LIN {X 0,Y 312.525,Z 361.177,A -85,B 0,C 180,E1 -15697.386,E2 -15697.386} C_VEL
LIN {X 0,Y 312.489,Z 361.185,A -85,B 0,C 180,E1 -15700.71,E2 -15700.71} C_VEL
LIN {X 0,Y 312.451,Z 361.181,A -85,B 0,C 180,E1 -15704.211,E2 -15704.211} C_VEL
LIN {X 0,Y 312.483,Z 361.184,A -85,B 0,C 180,E1 -15707.92,E2 -15707.92} C_VEL
LIN {X 0,Y 312.498,Z 361.177,A -85,B 0,C 180,E1 -15710.972,E2 -15710.972} C_VEL
LIN {X 0,Y 312.533,Z 361.179,A -85,B 0,C 180,E1 -15714.221,E2 -15714.221} C_VEL
LIN {X 0,Y 312.502,Z 361.178,A -85,B 0,C 180,E1 -15717.334,E2 -15717.334} C_VEL
LIN {X 0,Y 312.521,Z 361.179,A -85,B 0,C 180,E1 -15721.288,E2 -15721.288} C_VEL
LIN {X 0,Y 312.554,Z 361.175,A -85,B 0,C 180,E1 -15724.709,E2 -15724.709} C_VEL
LIN {X 0,Y 312.586,Z 361.17,A -85,B 0,C 180,E1 -15727.53,E2 -15727.53} C_VEL
LIN {X 0,Y 312.554,Z 361.175,A -85,B 0,C 180,E1 -15731.652,E2 -15731.652} C_VEL
LIN {X 0,Y 312.654,Z 361.162,A -85,B 0,C 180,E1 -15735.685,E2 -15735.685} C_VEL
LIN {X 0,Y 312.689,Z 361.158,A -85,B 0,C 180,E1 -15739.642,E2 -15739.642} C_VEL
LIN {X 0,Y 312.799,Z 361.146,A -85,B 0,C 180,E1 -15742.253,E2 -15742.253} C_VEL
LIN {X 0,Y 312.692,Z 361.158,A -85,B 0,C 180,E1 -15744.843,E2 -15744.843} C_VEL
LIN {X 0,Y 312.971,Z 361.126,A -85,B 0,C 180,E1 -15748.714,E2 -15748.714} C_VEL
LIN {X 0,Y 312.978,Z 361.123,A -85,B 0,C 180,E1 -15751.287,E2 -15751.287} C_VEL
LIN {X 0,Y 312.666,Z 361.158,A -85,B 0,C 180,E1 -15753.746,E2 -15753.746} C_VEL
LIN {X 0,Y 313.797,Z 364.207,A -85,B 0,C 180,E1 -15753.98,E2 -15753.98} C_VEL
LIN {X 0,Y 315.109,Z 366.459,A -85,B 0,C 180,E1 -15754.197,E2 -15754.197} C_VEL
LIN {X 0,Y 322.201,Z 378.936,A -85,B 0,C 180,E1 -15755.345,E2 -15755.345} C_VEL
LIN {X 0,Y 335.075,Z 404.668,A -85,B 0,C 180,E1 -15757.378,E2 -15757.378} C_VEL
LIN {X 0,Y 330.989,Z 518.086,A -85,B 0,C 180,E1 -15760.012,E2 -15760.012} C_VEL
LIN {X 0,Y 330.01,Z 533.872,A -85,B 0,C 180,E1 -15760.624,E2 -15760.624} C_VEL
LIN {X 0,Y 328.651,Z 549.395,A -85,B 0,C 180,E1 -15761.487,E2 -15761.487} C_VEL
LIN {X 0,Y 326.95,Z 564.144,A -85,B 0,C 180,E1 -15762.571,E2 -15762.571} C_VEL
LIN {X 0,Y 325.282,Z 576.901,A -85,B 0,C 180,E1 -15763.749,E2 -15763.749} C_VEL
LIN {X 0,Y 323.144,Z 590.398,A -85,B 0,C 180,E1 -15765.278,E2 -15765.278} C_VEL
LIN {X 0,Y 321,Z 602.964,A -85,B 0,C 180,E1 -15767.028,E2 -15767.028} C_VEL
LIN {X 0,Y 318.919,Z 614.479,A -85,B 0,C 180,E1 -15768.977,E2 -15768.977} C_VEL
LIN {X 0,Y 317.03,Z 624.528,A -85,B 0,C 180,E1 -15771.026,E2 -15771.026} C_VEL
LIN {X 0,Y 315.313,Z 633.751,A -85,B 0,C 180,E1 -15773.306,E2 -15773.306} C_VEL
LIN {X 0,Y 313.823,Z 641.736,A -85,B 0,C 180,E1 -15775.715,E2 -15775.715} C_VEL
LIN {X 0,Y 312.703,Z 648.292,A -85,B 0,C 180,E1 -15778.163,E2 -15778.163} C_VEL
LIN {X 0,Y 311.992,Z 652.989,A -85,B 0,C 180,E1 -15780.373,E2 -15780.373} C_VEL
LIN {X 0,Y 311.387,Z 657.033,A -85,B 0,C 180,E1 -15782.799,E2 -15782.799} C_VEL
LIN {X 0,Y 310.853,Z 660.262,A -85,B 0,C 180,E1 -15785.519,E2 -15785.519} C_VEL
LIN {X 0,Y 310.67,Z 661.884,A -85,B 0,C 180,E1 -15787.648,E2 -15787.648} C_VEL
LIN {X 0,Y 310.638,Z 662.675,A -85,B 0,C 180,E1 -15789.714,E2 -15789.714} C_VEL
LIN {X 0,Y 310.68,Z 662.765,A -85,B 0,C 180,E1 -15791.711,E2 -15791.711} C_VEL
LIN {X 0,Y 310.986,Z 661.766,A -85,B 0,C 180,E1 -15794.474,E2 -15794.474} C_VEL
LIN {X 0,Y 311.302,Z 660.45,A -85,B 0,C 180,E1 -15796.257,E2 -15796.257} C_VEL
LIN {X 0,Y 312.085,Z 656.982,A -85,B 0,C 180,E1 -15799.226,E2 -15799.226} C_VEL
LIN {X 0,Y 312.245,Z 656.181,A -85,B 0,C 180,E1 -15799.738,E2 -15799.738} C_VEL
LIN {X 0,Y 311.958,Z 654.592,A -85,B 0,C 180,E1 -15800.782,E2 -15800.782} C_VEL
LIN {X 0,Y 309.828,Z 651.885,A -85,B 0,C 180,E1 -15802.5,E2 -15802.5} C_VEL
LIN {X 0,Y 307.865,Z 648.675,A -85,B 0,C 180,E1 -15804.206,E2 -15804.206} C_VEL
LIN {X 0,Y 307.837,Z 646.264,A -85,B 0,C 180,E1 -15805.211,E2 -15805.211} C_VEL
LIN {X 0,Y 309.567,Z 639.569,A -85,B 0,C 180,E1 -15807.567,E2 -15807.567} C_VEL
LIN {X 0,Y 311.823,Z 630.956,A -85,B 0,C 180,E1 -15810.021,E2 -15810.021} C_VEL
LIN {X 0,Y 314.423,Z 621.191,A -85,B 0,C 180,E1 -15812.277,E2 -15812.277} C_VEL
LIN {X 0,Y 317.078,Z 610.167,A -85,B 0,C 180,E1 -15814.379,E2 -15814.379} C_VEL
LIN {X 0,Y 319.674,Z 598.716,A -85,B 0,C 180,E1 -15816.173,E2 -15816.173} C_VEL
LIN {X 0,Y 322.229,Z 586.6,A -85,B 0,C 180,E1 -15817.73,E2 -15817.73} C_VEL
LIN {X 0,Y 324.848,Z 572.636,A -85,B 0,C 180,E1 -15819.188,E2 -15819.188} C_VEL
LIN {X 0,Y 326.941,Z 558.599,A -85,B 0,C 180,E1 -15820.365,E2 -15820.365} C_VEL
LIN {X 0,Y 328.688,Z 544.34,A -85,B 0,C 180,E1 -15821.292,E2 -15821.292} C_VEL
LIN {X 0,Y 330.129,Z 528.83,A -85,B 0,C 180,E1 -15822.04,E2 -15822.04} C_VEL
LIN {X 0,Y 331.077,Z 513.629,A -85,B 0,C 180,E1 -15822.523,E2 -15822.523} C_VEL
LIN {X 0,Y 335.904,Z 411.379,A -85,B 0,C 180,E1 -15824.997,E2 -15824.997} C_VEL
LIN {X 0,Y 329.841,Z 399.642,A -85,B 0,C 180,E1 -15826.309,E2 -15826.309} C_VEL
LIN {X 0,Y 321.07,Z 385.074,A -85,B 0,C 180,E1 -15828.31,E2 -15828.31} C_VEL
LIN {X 0,Y 314.835,Z 375.782,A -85,B 0,C 180,E1 -15829.839,E2 -15829.839} C_VEL
LIN {X 0,Y 311.604,Z 371.252,A -85,B 0,C 180,E1 -15830.682,E2 -15830.682} C_VEL
LIN {X 0,Y 309.38,Z 367.982,A -85,B 0,C 180,E1 -15831.288,E2 -15831.288} C_VEL
LIN {X 0,Y 308.675,Z 366.924,A -85,B 0,C 180,E1 -15831.487,E2 -15831.487} C_VEL
LIN {X 0,Y 306.652,Z 364.665,A -85,B 0,C 180,E1 -15832.04,E2 -15832.04} C_VEL
LIN {X 0,Y 305.758,Z 362.023,A -85,B 0,C 180,E1 -15832.405,E2 -15832.405} C_VEL
LIN {X 0,Y 305.858,Z 362.008,A -85,B 0,C 180,E1 -15837.366,E2 -15837.366} C_VEL
LIN {X 0,Y 306.012,Z 361.989,A -85,B 0,C 180,E1 -15840,E2 -15840} C_VEL
LIN {X 0,Y 305.882,Z 362.006,A -85,B 0,C 180,E1 -15842.633,E2 -15842.633} C_VEL
LIN {X 0,Y 305.79,Z 362.017,A -85,B 0,C 180,E1 -15846.598,E2 -15846.598} C_VEL
LIN {X 0,Y 305.697,Z 362.029,A -85,B 0,C 180,E1 -15849.26,E2 -15849.26} C_VEL
LIN {X 0,Y 305.589,Z 362.038,A -85,B 0,C 180,E1 -15853.296,E2 -15853.296} C_VEL
LIN {X 0,Y 305.554,Z 362.041,A -85,B 0,C 180,E1 -15856.022,E2 -15856.022} C_VEL
LIN {X 0,Y 305.563,Z 362.043,A -85,B 0,C 180,E1 -15859.436,E2 -15859.436} C_VEL
LIN {X 0,Y 305.493,Z 362.058,A -85,B 0,C 180,E1 -15863.041,E2 -15863.041} C_VEL
LIN {X 0,Y 305.55,Z 362.05,A -85,B 0,C 180,E1 -15866.227,E2 -15866.227} C_VEL
LIN {X 0,Y 305.498,Z 362.054,A -85,B 0,C 180,E1 -15869.049,E2 -15869.049} C_VEL
LIN {X 0,Y 305.467,Z 362.063,A -85,B 0,C 180,E1 -15873.516,E2 -15873.516} C_VEL
LIN {X 0,Y 305.497,Z 362.055,A -85,B 0,C 180,E1 -15876.736,E2 -15876.736} C_VEL
LIN {X 0,Y 305.456,Z 362.063,A -85,B 0,C 180,E1 -15880.599,E2 -15880.599} C_VEL
LIN {X 0,Y 305.453,Z 362.134,A -85,B 0,C 180,E1 -15881.768,E2 -15881.768} C_VEL
LIN {X 0,Y 308.493,Z 370.686,A -85,B 0,C 180,E1 -15885.391,E2 -15885.391} C_VEL
LIN {X 0,Y 311.562,Z 380.053,A -85,B 0,C 180,E1 -15888.832,E2 -15888.832} C_VEL
LIN {X 0,Y 314.609,Z 385.314,A -85,B 0,C 180,E1 -15889.657,E2 -15889.657} C_VEL
LIN {X 0,Y 321.104,Z 396.951,A -85,B 0,C 180,E1 -15891.302,E2 -15891.302} C_VEL
LIN {X 0,Y 327.272,Z 409.327,A -85,B 0,C 180,E1 -15892.78,E2 -15892.78} C_VEL
LIN {X 0,Y 331.591,Z 419.42,A -85,B 0,C 180,E1 -15893.794,E2 -15893.794} C_VEL
LIN {X 0,Y 334.763,Z 442.582,A -85,B 0,C 180,E1 -15894.992,E2 -15894.992} C_VEL
LIN {X 0,Y 329.679,Z 550.26,A -85,B 0,C 180,E1 -15897.614,E2 -15897.614} C_VEL
LIN {X 0,Y 328.139,Z 566.262,A -85,B 0,C 180,E1 -15898.214,E2 -15898.214} C_VEL
LIN {X 0,Y 326.128,Z 581.586,A -85,B 0,C 180,E1 -15899.035,E2 -15899.035} C_VEL
LIN {X 0,Y 323.802,Z 595.93,A -85,B 0,C 180,E1 -15900.052,E2 -15900.052} C_VEL
LIN {X 0,Y 321.345,Z 609.142,A -85,B 0,C 180,E1 -15901.239,E2 -15901.239} C_VEL
LIN {X 0,Y 318.545,Z 622.691,A -85,B 0,C 180,E1 -15902.754,E2 -15902.754} C_VEL
LIN {X 0,Y 315.712,Z 635.085,A -85,B 0,C 180,E1 -15904.449,E2 -15904.449} C_VEL
LIN {X 0,Y 312.807,Z 647.316,A -85,B 0,C 180,E1 -15906.496,E2 -15906.496} C_VEL
LIN {X 0,Y 310.294,Z 658.302,A -85,B 0,C 180,E1 -15908.752,E2 -15908.752} C_VEL
LIN {X 0,Y 308.125,Z 667.5,A -85,B 0,C 180,E1 -15911.032,E2 -15911.032} C_VEL
LIN {X 0,Y 306.463,Z 675.179,A -85,B 0,C 180,E1 -15913.341,E2 -15913.341} C_VEL
LIN {X 0,Y 305.112,Z 682.376,A -85,B 0,C 180,E1 -15916.003,E2 -15916.003} C_VEL
LIN {X 0,Y 304.259,Z 688.089,A -85,B 0,C 180,E1 -15918.676,E2 -15918.676} C_VEL
LIN {X 0,Y 303.897,Z 691.49,A -85,B 0,C 180,E1 -15920.683,E2 -15920.683} C_VEL
LIN {X 0,Y 303.719,Z 694.922,A -85,B 0,C 180,E1 -15923.355,E2 -15923.355} C_VEL
LIN {X 0,Y 303.733,Z 697.078,A -85,B 0,C 180,E1 -15926.019,E2 -15926.019} C_VEL
LIN {X 0,Y 303.826,Z 698.028,A -85,B 0,C 180,E1 -15928.674,E2 -15928.674} C_VEL
LIN {X 0,Y 303.935,Z 698.061,A -85,B 0,C 180,E1 -15929.999,E2 -15929.999} C_VEL
LIN {X 0,Y 303.759,Z 697.203,A -85,B 0,C 180,E1 -15932.652,E2 -15932.652} C_VEL
LIN {X 0,Y 303.722,Z 695.129,A -85,B 0,C 180,E1 -15935.31,E2 -15935.31} C_VEL
LIN {X 0,Y 303.803,Z 691.785,A -85,B 0,C 180,E1 -15937.978,E2 -15937.978} C_VEL
LIN {X 0,Y 304.059,Z 687.063,A -85,B 0,C 180,E1 -15940.655,E2 -15940.655} C_VEL
LIN {X 0,Y 304.782,Z 680.879,A -85,B 0,C 180,E1 -15943.331,E2 -15943.331} C_VEL
LIN {X 0,Y 305.951,Z 673.077,A -85,B 0,C 180,E1 -15946,E2 -15946} C_VEL
LIN {X 0,Y 307.348,Z 664.692,A -85,B 0,C 180,E1 -15948.325,E2 -15948.325} C_VEL
LIN {X 0,Y 309.283,Z 654.625,A -85,B 0,C 180,E1 -15950.622,E2 -15950.622} C_VEL
LIN {X 0,Y 311.152,Z 644.275,A -85,B 0,C 180,E1 -15952.58,E2 -15952.58} C_VEL
LIN {X 0,Y 313.211,Z 633.065,A -85,B 0,C 180,E1 -15954.349,E2 -15954.349} C_VEL
LIN {X 0,Y 315.421,Z 620.977,A -85,B 0,C 180,E1 -15955.929,E2 -15955.929} C_VEL
LIN {X 0,Y 317.659,Z 607.911,A -85,B 0,C 180,E1 -15957.327,E2 -15957.327} C_VEL
LIN {X 0,Y 319.827,Z 593.492,A -85,B 0,C 180,E1 -15958.564,E2 -15958.564} C_VEL
LIN {X 0,Y 321.489,Z 580.177,A -85,B 0,C 180,E1 -15959.463,E2 -15959.463} C_VEL
LIN {X 0,Y 323.084,Z 564.612,A -85,B 0,C 180,E1 -15960.245,E2 -15960.245} C_VEL
LIN {X 0,Y 324.137,Z 549.447,A -85,B 0,C 180,E1 -15960.767,E2 -15960.767} C_VEL
LIN {X 0,Y 328.19,Z 442.647,A -85,B 0,C 180,E1 -15963.277,E2 -15963.277} C_VEL
LIN {X 0,Y 324.682,Z 419.062,A -85,B 0,C 180,E1 -15964.279,E2 -15964.279} C_VEL
LIN {X 0,Y 323.2,Z 411.08,A -85,B 0,C 180,E1 -15964.658,E2 -15964.658} C_VEL
LIN {X 0,Y 314.936,Z 392.022,A -85,B 0,C 180,E1 -15966.101,E2 -15966.101} C_VEL
LIN {X 0,Y 311.738,Z 384.895,A -85,B 0,C 180,E1 -15966.705,E2 -15966.705} C_VEL
LIN {X 0,Y 308.469,Z 372.592,A -85,B 0,C 180,E1 -15969.961,E2 -15969.961} C_VEL
LIN {X 0,Y 305.432,Z 362.068,A -85,B 0,C 180,E1 -15972.973,E2 -15972.973} C_VEL
LIN {X 0,Y 305.456,Z 362.057,A -85,B 0,C 180,E1 -15977.413,E2 -15977.413} C_VEL
LIN {X 0,Y 305.472,Z 362.054,A -85,B 0,C 180,E1 -15981.597,E2 -15981.597} C_VEL
LIN {X 0,Y 305.459,Z 362.065,A -85,B 0,C 180,E1 -15984.887,E2 -15984.887} C_VEL
LIN {X 0,Y 305.448,Z 362.061,A -85,B 0,C 180,E1 -15988.355,E2 -15988.355} C_VEL
LIN {X 0,Y 305.517,Z 362.055,A -85,B 0,C 180,E1 -15991.114,E2 -15991.114} C_VEL
LIN {X 0,Y 305.568,Z 362.043,A -85,B 0,C 180,E1 -15994.088,E2 -15994.088} C_VEL
LIN {X 0,Y 305.497,Z 362.053,A -85,B 0,C 180,E1 -15998.403,E2 -15998.403} C_VEL
LIN {X 0,Y 305.586,Z 362.044,A -85,B 0,C 180,E1 -16001.218,E2 -16001.218} C_VEL
LIN {X 0,Y 305.646,Z 362.036,A -85,B 0,C 180,E1 -16005.349,E2 -16005.349} C_VEL
LIN {X 0,Y 305.635,Z 362.025,A -85,B 0,C 180,E1 -16009.4,E2 -16009.4} C_VEL
LIN {X 0,Y 305.805,Z 362.012,A -85,B 0,C 180,E1 -16012.075,E2 -16012.075} C_VEL
LIN {X 0,Y 305.685,Z 362.033,A -85,B 0,C 180,E1 -16014.724,E2 -16014.724} C_VEL
LIN {X 0,Y 305.955,Z 361.991,A -85,B 0,C 180,E1 -16018.684,E2 -16018.684} C_VEL
LIN {X 0,Y 305.955,Z 361.998,A -85,B 0,C 180,E1 -16021.317,E2 -16021.317} C_VEL
LIN {X 0,Y 305.85,Z 362.005,A -85,B 0,C 180,E1 -16026.598,E2 -16026.598} C_VEL
LIN {X 0,Y 305.734,Z 362.024,A -85,B 0,C 180,E1 -16029.26,E2 -16029.26} C_VEL
LIN {X 0,Y 305.587,Z 362.042,A -85,B 0,C 180,E1 -16033.297,E2 -16033.297} C_VEL
LIN {X 0,Y 305.592,Z 362.034,A -85,B 0,C 180,E1 -16036.021,E2 -16036.021} C_VEL
LIN {X 0,Y 305.574,Z 362.043,A -85,B 0,C 180,E1 -16039.445,E2 -16039.445} C_VEL
LIN {X 0,Y 305.484,Z 362.054,A -85,B 0,C 180,E1 -16043.04,E2 -16043.04} C_VEL
LIN {X 0,Y 305.525,Z 362.041,A -85,B 0,C 180,E1 -16046.22,E2 -16046.22} C_VEL
LIN {X 0,Y 305.495,Z 362.056,A -85,B 0,C 180,E1 -16049.051,E2 -16049.051} C_VEL
LIN {X 0,Y 305.464,Z 362.052,A -85,B 0,C 180,E1 -16053.518,E2 -16053.518} C_VEL
LIN {X 0,Y 305.474,Z 362.056,A -85,B 0,C 180,E1 -16056.74,E2 -16056.74} C_VEL
LIN {X 0,Y 305.454,Z 362.062,A -85,B 0,C 180,E1 -16060.601,E2 -16060.601} C_VEL
LIN {X 0,Y 305.425,Z 362.053,A -85,B 0,C 180,E1 -16063.656,E2 -16063.656} C_VEL
LIN {X 0,Y 305.454,Z 362.059,A -85,B 0,C 180,E1 -16067.415,E2 -16067.415} C_VEL
LIN {X 0,Y 305.467,Z 362.05,A -85,B 0,C 180,E1 -16071.597,E2 -16071.597} C_VEL
LIN {X 0,Y 305.463,Z 362.06,A -85,B 0,C 180,E1 -16074.888,E2 -16074.888} C_VEL
LIN {X 0,Y 305.443,Z 362.058,A -85,B 0,C 180,E1 -16078.359,E2 -16078.359} C_VEL
LIN {X 0,Y 305.488,Z 362.056,A -85,B 0,C 180,E1 -16081.111,E2 -16081.111} C_VEL
LIN {X 0,Y 305.506,Z 362.052,A -85,B 0,C 180,E1 -16084.083,E2 -16084.083} C_VEL
LIN {X 0,Y 305.49,Z 362.056,A -85,B 0,C 180,E1 -16088.403,E2 -16088.403} C_VEL
LIN {X 0,Y 305.512,Z 362.052,A -85,B 0,C 180,E1 -16091.213,E2 -16091.213} C_VEL
LIN {X 0,Y 305.582,Z 362.043,A -85,B 0,C 180,E1 -16095.346,E2 -16095.346} C_VEL
LIN {X 0,Y 305.627,Z 362.037,A -85,B 0,C 180,E1 -16099.4,E2 -16099.4} C_VEL
LIN {X 0,Y 305.75,Z 362.023,A -85,B 0,C 180,E1 -16102.073,E2 -16102.073} C_VEL
LIN {X 0,Y 305.662,Z 362.034,A -85,B 0,C 180,E1 -16104.724,E2 -16104.724} C_VEL
LIN {X 0,Y 305.939,Z 362.002,A -85,B 0,C 180,E1 -16108.684,E2 -16108.684} C_VEL
LIN {X 0,Y 305.946,Z 362,A -85,B 0,C 180,E1 -16111.317,E2 -16111.317} C_VEL
LIN {X 0,Y 305.773,Z 362.014,A -85,B 0,C 180,E1 -16112.932,E2 -16112.932} C_VEL
LIN {X 0,Y 306.841,Z 365.057,A -85,B 0,C 180,E1 -16113.18,E2 -16113.18} C_VEL
LIN {X 0,Y 316.889,Z 382.866,A -85,B 0,C 180,E1 -16114.879,E2 -16114.879} C_VEL
LIN {X 0,Y 328.783,Z 406.691,A -85,B 0,C 180,E1 -16116.808,E2 -16116.808} C_VEL
LIN {X 0,Y 324.637,Z 518.559,A -85,B 0,C 180,E1 -16119.463,E2 -16119.463} C_VEL
LIN {X 0,Y 323.669,Z 533.986,A -85,B 0,C 180,E1 -16120.07,E2 -16120.07} C_VEL
LIN {X 0,Y 322.334,Z 549.035,A -85,B 0,C 180,E1 -16120.913,E2 -16120.913} C_VEL
LIN {X 0,Y 320.545,Z 564.038,A -85,B 0,C 180,E1 -16122.023,E2 -16122.023} C_VEL
LIN {X 0,Y 318.572,Z 578.392,A -85,B 0,C 180,E1 -16123.384,E2 -16123.384} C_VEL
LIN {X 0,Y 316.352,Z 591.876,A -85,B 0,C 180,E1 -16124.967,E2 -16124.967} C_VEL
LIN {X 0,Y 314.197,Z 604.035,A -85,B 0,C 180,E1 -16126.716,E2 -16126.716} C_VEL
LIN {X 0,Y 312.407,Z 613.648,A -85,B 0,C 180,E1 -16128.358,E2 -16128.358} C_VEL
LIN {X 0,Y 310.328,Z 624.354,A -85,B 0,C 180,E1 -16130.551,E2 -16130.551} C_VEL
LIN {X 0,Y 308.577,Z 633.32,A -85,B 0,C 180,E1 -16132.78,E2 -16132.78} C_VEL
LIN {X 0,Y 307.109,Z 640.854,A -85,B 0,C 180,E1 -16135.048,E2 -16135.048} C_VEL
LIN {X 0,Y 305.932,Z 647.161,A -85,B 0,C 180,E1 -16137.352,E2 -16137.352} C_VEL
LIN {X 0,Y 305.111,Z 652.347,A -85,B 0,C 180,E1 -16139.685,E2 -16139.685} C_VEL
LIN {X 0,Y 304.484,Z 656.53,A -85,B 0,C 180,E1 -16142.065,E2 -16142.065} C_VEL
LIN {X 0,Y 304.082,Z 658.757,A -85,B 0,C 180,E1 -16143.69,E2 -16143.69} C_VEL
LIN {X 0,Y 303.717,Z 661.043,A -85,B 0,C 180,E1 -16145.913,E2 -16145.913} C_VEL
LIN {X 0,Y 303.558,Z 662.756,A -85,B 0,C 180,E1 -16148.691,E2 -16148.691} C_VEL
LIN {X 0,Y 303.564,Z 663.194,A -85,B 0,C 180,E1 -16150.41,E2 -16150.41} C_VEL
LIN {X 0,Y 303.632,Z 663.156,A -85,B 0,C 180,E1 -16152.209,E2 -16152.209} C_VEL
LIN {X 0,Y 303.848,Z 662.447,A -85,B 0,C 180,E1 -16154.189,E2 -16154.189} C_VEL
LIN {X 0,Y 304.184,Z 661.159,A -85,B 0,C 180,E1 -16156.121,E2 -16156.121} C_VEL
LIN {X 0,Y 304.647,Z 659.329,A -85,B 0,C 180,E1 -16158.008,E2 -16158.008} C_VEL
LIN {X 0,Y 305.5,Z 655.63,A -85,B 0,C 180,E1 -16160.679,E2 -16160.679} C_VEL
LIN {X 0,Y 306.768,Z 650.421,A -85,B 0,C 180,E1 -16163.44,E2 -16163.44} C_VEL
LIN {X 0,Y 307.837,Z 646.264,A -85,B 0,C 180,E1 -16165.211,E2 -16165.211} C_VEL
LIN {X 0,Y 307.873,Z 643.766,A -85,B 0,C 180,E1 -16166.201,E2 -16166.201} C_VEL
LIN {X 0,Y 306.311,Z 639.635,A -85,B 0,C 180,E1 -16167.855,E2 -16167.855} C_VEL
LIN {X 0,Y 304.897,Z 635.081,A -85,B 0,C 180,E1 -16169.489,E2 -16169.489} C_VEL
LIN {X 0,Y 305.162,Z 631.888,A -85,B 0,C 180,E1 -16170.429,E2 -16170.429} C_VEL
LIN {X 0,Y 308.019,Z 621.685,A -85,B 0,C 180,E1 -16172.856,E2 -16172.856} C_VEL
LIN {X 0,Y 310.803,Z 610.698,A -85,B 0,C 180,E1 -16174.989,E2 -16174.989} C_VEL
LIN {X 0,Y 313.499,Z 599.334,A -85,B 0,C 180,E1 -16176.801,E2 -16176.801} C_VEL
LIN {X 0,Y 316.402,Z 586.157,A -85,B 0,C 180,E1 -16178.512,E2 -16178.512} C_VEL
LIN {X 0,Y 319.042,Z 572.446,A -85,B 0,C 180,E1 -16179.951,E2 -16179.951} C_VEL
LIN {X 0,Y 321.141,Z 559.097,A -85,B 0,C 180,E1 -16181.085,E2 -16181.085} C_VEL
LIN {X 0,Y 323.112,Z 543.453,A -85,B 0,C 180,E1 -16182.107,E2 -16182.107} C_VEL
LIN {X 0,Y 324.532,Z 528.086,A -85,B 0,C 180,E1 -16182.837,E2 -16182.837} C_VEL
LIN {X 0,Y 325.566,Z 512.416,A -85,B 0,C 180,E1 -16183.315,E2 -16183.315} C_VEL
LIN {X 0,Y 330.404,Z 413.808,A -85,B 0,C 180,E1 -16185.752,E2 -16185.752} C_VEL
LIN {X 0,Y 324.344,Z 402.299,A -85,B 0,C 180,E1 -16187.121,E2 -16187.121} C_VEL
LIN {X 0,Y 316.457,Z 389.025,A -85,B 0,C 180,E1 -16189.022,E2 -16189.022} C_VEL
LIN {X 0,Y 310.796,Z 380.655,A -85,B 0,C 180,E1 -16190.475,E2 -16190.475} C_VEL
LIN {X 0,Y 308.04,Z 376.701,A -85,B 0,C 180,E1 -16191.222,E2 -16191.222} C_VEL
LIN {X 0,Y 305.121,Z 372.518,A -85,B 0,C 180,E1 -16192.056,E2 -16192.056} C_VEL
LIN {X 0,Y 302.886,Z 369.527,A -85,B 0,C 180,E1 -16192.709,E2 -16192.709} C_VEL
LIN {X 0,Y 302.03,Z 368.043,A -85,B 0,C 180,E1 -16192.983,E2 -16192.983} C_VEL
LIN {X 0,Y 299.775,Z 365.827,A -85,B 0,C 180,E1 -16193.648,E2 -16193.648} C_VEL
LIN {X 0,Y 298.79,Z 363.526,A -85,B 0,C 180,E1 -16194.008,E2 -16194.008} C_VEL
LIN {X 0,Y 298.67,Z 362.908,A -85,B 0,C 180,E1 -16194.091,E2 -16194.091} C_VEL
LIN {X 0,Y 298.916,Z 362.876,A -85,B 0,C 180,E1 -16198.652,E2 -16198.652} C_VEL
LIN {X 0,Y 298.92,Z 362.873,A -85,B 0,C 180,E1 -16201.347,E2 -16201.347} C_VEL
LIN {X 0,Y 298.638,Z 362.908,A -85,B 0,C 180,E1 -16205.401,E2 -16205.401} C_VEL
LIN {X 0,Y 298.71,Z 362.903,A -85,B 0,C 180,E1 -16208.819,E2 -16208.819} C_VEL
LIN {X 0,Y 298.548,Z 362.917,A -85,B 0,C 180,E1 -16213.615,E2 -16213.615} C_VEL
LIN {X 0,Y 298.489,Z 362.923,A -85,B 0,C 180,E1 -16216.412,E2 -16216.412} C_VEL
LIN {X 0,Y 298.501,Z 362.925,A -85,B 0,C 180,E1 -16219.647,E2 -16219.647} C_VEL
LIN {X 0,Y 298.46,Z 362.93,A -85,B 0,C 180,E1 -16223.597,E2 -16223.597} C_VEL
LIN {X 0,Y 298.491,Z 362.926,A -85,B 0,C 180,E1 -16226.574,E2 -16226.574} C_VEL
LIN {X 0,Y 298.423,Z 362.932,A -85,B 0,C 180,E1 -16229.64,E2 -16229.64} C_VEL
LIN {X 0,Y 298.397,Z 362.937,A -85,B 0,C 180,E1 -16232.799,E2 -16232.799} C_VEL
LIN {X 0,Y 298.466,Z 362.931,A -85,B 0,C 180,E1 -16236.812,E2 -16236.812} C_VEL
LIN {X 0,Y 298.421,Z 362.951,A -85,B 0,C 180,E1 -16240.143,E2 -16240.143} C_VEL
LIN {X 0,Y 301.067,Z 370.515,A -85,B 0,C 180,E1 -16243.642,E2 -16243.642} C_VEL
LIN {X 0,Y 303.349,Z 377.253,A -85,B 0,C 180,E1 -16246.385,E2 -16246.385} C_VEL
LIN {X 0,Y 304.157,Z 379.526,A -85,B 0,C 180,E1 -16247.191,E2 -16247.191} C_VEL
LIN {X 0,Y 307.599,Z 385.003,A -85,B 0,C 180,E1 -16248.194,E2 -16248.194} C_VEL
LIN {X 0,Y 312.48,Z 393.558,A -85,B 0,C 180,E1 -16249.551,E2 -16249.551} C_VEL
LIN {X 0,Y 318.528,Z 404.794,A -85,B 0,C 180,E1 -16251.118,E2 -16251.118} C_VEL
LIN {X 0,Y 324.473,Z 417.574,A -85,B 0,C 180,E1 -16252.601,E2 -16252.601} C_VEL
LIN {X 0,Y 326.593,Z 422.93,A -85,B 0,C 180,E1 -16253.125,E2 -16253.125} C_VEL
LIN {X 0,Y 329.297,Z 443.898,A -85,B 0,C 180,E1 -16254.237,E2 -16254.237} C_VEL
LIN {X 0,Y 324.08,Z 549.494,A -85,B 0,C 180,E1 -16256.845,E2 -16256.845} C_VEL
LIN {X 0,Y 322.452,Z 565.528,A -85,B 0,C 180,E1 -16257.447,E2 -16257.447} C_VEL
LIN {X 0,Y 320.468,Z 580.295,A -85,B 0,C 180,E1 -16258.242,E2 -16258.242} C_VEL
LIN {X 0,Y 317.987,Z 594.759,A -85,B 0,C 180,E1 -16259.262,E2 -16259.262} C_VEL
LIN {X 0,Y 315.17,Z 609.522,A -85,B 0,C 180,E1 -16260.621,E2 -16260.621} C_VEL
LIN {X 0,Y 312.243,Z 622.927,A -85,B 0,C 180,E1 -16262.157,E2 -16262.157} C_VEL
LIN {X 0,Y 309.303,Z 635.222,A -85,B 0,C 180,E1 -16263.88,E2 -16263.88} C_VEL
LIN {X 0,Y 306.704,Z 645.623,A -85,B 0,C 180,E1 -16265.64,E2 -16265.64} C_VEL
LIN {X 0,Y 303.904,Z 656.89,A -85,B 0,C 180,E1 -16267.945,E2 -16267.945} C_VEL
LIN {X 0,Y 301.664,Z 666.142,A -85,B 0,C 180,E1 -16270.256,E2 -16270.256} C_VEL
LIN {X 0,Y 299.584,Z 675.002,A -85,B 0,C 180,E1 -16272.947,E2 -16272.947} C_VEL
LIN {X 0,Y 298.158,Z 682.156,A -85,B 0,C 180,E1 -16275.67,E2 -16275.67} C_VEL
LIN {X 0,Y 297.217,Z 687.815,A -85,B 0,C 180,E1 -16278.404,E2 -16278.404} C_VEL
LIN {X 0,Y 296.828,Z 691.17,A -85,B 0,C 180,E1 -16280.459,E2 -16280.459} C_VEL
LIN {X 0,Y 296.635,Z 694.567,A -85,B 0,C 180,E1 -16283.196,E2 -16283.196} C_VEL
LIN {X 0,Y 296.642,Z 696.707,A -85,B 0,C 180,E1 -16285.924,E2 -16285.924} C_VEL
LIN {X 0,Y 296.732,Z 697.623,A -85,B 0,C 180,E1 -16288.642,E2 -16288.642} C_VEL
LIN {X 0,Y 296.846,Z 697.638,A -85,B 0,C 180,E1 -16289.999,E2 -16289.999} C_VEL
LIN {X 0,Y 296.679,Z 696.742,A -85,B 0,C 180,E1 -16292.715,E2 -16292.715} C_VEL
LIN {X 0,Y 296.64,Z 694.627,A -85,B 0,C 180,E1 -16295.437,E2 -16295.437} C_VEL
LIN {X 0,Y 296.746,Z 691.241,A -85,B 0,C 180,E1 -16298.169,E2 -16298.169} C_VEL
LIN {X 0,Y 297.019,Z 686.483,A -85,B 0,C 180,E1 -16300.911,E2 -16300.911} C_VEL
LIN {X 0,Y 297.792,Z 680.25,A -85,B 0,C 180,E1 -16303.65,E2 -16303.65} C_VEL
LIN {X 0,Y 299.046,Z 672.378,A -85,B 0,C 180,E1 -16306.38,E2 -16306.38} C_VEL
LIN {X 0,Y 300.509,Z 663.943,A -85,B 0,C 180,E1 -16308.757,E2 -16308.757} C_VEL
LIN {X 0,Y 302.555,Z 653.798,A -85,B 0,C 180,E1 -16311.102,E2 -16311.102} C_VEL
LIN {X 0,Y 304.503,Z 643.37,A -85,B 0,C 180,E1 -16313.101,E2 -16313.101} C_VEL
LIN {X 0,Y 306.951,Z 630.979,A -85,B 0,C 180,E1 -16315.06,E2 -16315.06} C_VEL
LIN {X 0,Y 309.277,Z 618.549,A -85,B 0,C 180,E1 -16316.666,E2 -16316.666} C_VEL
LIN {X 0,Y 311.59,Z 605.031,A -85,B 0,C 180,E1 -16318.088,E2 -16318.088} C_VEL
LIN {X 0,Y 313.603,Z 591.232,A -85,B 0,C 180,E1 -16319.253,E2 -16319.253} C_VEL
LIN {X 0,Y 315.407,Z 577.052,A -85,B 0,C 180,E1 -16320.181,E2 -16320.181} C_VEL
LIN {X 0,Y 316.923,Z 562.237,A -85,B 0,C 180,E1 -16320.897,E2 -16320.897} C_VEL
LIN {X 0,Y 317.918,Z 547.341,A -85,B 0,C 180,E1 -16321.391,E2 -16321.391} C_VEL
LIN {X 0,Y 321.999,Z 442.984,A -85,B 0,C 180,E1 -16323.887,E2 -16323.887} C_VEL
LIN {X 0,Y 317.554,Z 414.319,A -85,B 0,C 180,E1 -16325.166,E2 -16325.166} C_VEL
LIN {X 0,Y 309.597,Z 395.873,A -85,B 0,C 180,E1 -16326.591,E2 -16326.591} C_VEL
LIN {X 0,Y 304.386,Z 384.503,A -85,B 0,C 180,E1 -16327.572,E2 -16327.572} C_VEL
LIN {X 0,Y 301.233,Z 372.773,A -85,B 0,C 180,E1 -16330.787,E2 -16330.787} C_VEL
LIN {X 0,Y 298.402,Z 362.944,A -85,B 0,C 180,E1 -16333.71,E2 -16333.71} C_VEL
LIN {X 0,Y 298.399,Z 362.941,A -85,B 0,C 180,E1 -16336.921,E2 -16336.921} C_VEL
LIN {X 0,Y 298.4,Z 362.938,A -85,B 0,C 180,E1 -16341.006,E2 -16341.006} C_VEL
LIN {X 0,Y 298.415,Z 362.94,A -85,B 0,C 180,E1 -16343.93,E2 -16343.93} C_VEL
LIN {X 0,Y 298.392,Z 362.94,A -85,B 0,C 180,E1 -16347.983,E2 -16347.983} C_VEL
LIN {X 0,Y 298.46,Z 362.932,A -85,B 0,C 180,E1 -16351.904,E2 -16351.904} C_VEL
LIN {X 0,Y 298.482,Z 362.929,A -85,B 0,C 180,E1 -16354.924,E2 -16354.924} C_VEL
LIN {X 0,Y 298.446,Z 362.936,A -85,B 0,C 180,E1 -16359.315,E2 -16359.315} C_VEL
LIN {X 0,Y 298.534,Z 362.919,A -85,B 0,C 180,E1 -16362.18,E2 -16362.18} C_VEL
LIN {X 0,Y 298.59,Z 362.918,A -85,B 0,C 180,E1 -16364.995,E2 -16364.995} C_VEL
LIN {X 0,Y 298.59,Z 362.9,A -85,B 0,C 180,E1 -16369.147,E2 -16369.147} C_VEL
LIN {X 0,Y 298.751,Z 362.89,A -85,B 0,C 180,E1 -16371.886,E2 -16371.886} C_VEL
LIN {X 0,Y 298.655,Z 362.908,A -85,B 0,C 180,E1 -16374.599,E2 -16374.599} C_VEL
LIN {X 0,Y 298.921,Z 362.866,A -85,B 0,C 180,E1 -16378.653,E2 -16378.653} C_VEL
LIN {X 0,Y 298.921,Z 362.874,A -85,B 0,C 180,E1 -16381.348,E2 -16381.348} C_VEL
LIN {X 0,Y 298.796,Z 362.882,A -85,B 0,C 180,E1 -16386.754,E2 -16386.754} C_VEL
LIN {X 0,Y 298.678,Z 362.901,A -85,B 0,C 180,E1 -16389.481,E2 -16389.481} C_VEL
LIN {X 0,Y 298.55,Z 362.917,A -85,B 0,C 180,E1 -16393.616,E2 -16393.616} C_VEL
LIN {X 0,Y 298.547,Z 362.911,A -85,B 0,C 180,E1 -16396.409,E2 -16396.409} C_VEL
LIN {X 0,Y 298.508,Z 362.923,A -85,B 0,C 180,E1 -16399.655,E2 -16399.655} C_VEL
LIN {X 0,Y 298.427,Z 362.93,A -85,B 0,C 180,E1 -16403.601,E2 -16403.601} C_VEL
LIN {X 0,Y 298.484,Z 362.919,A -85,B 0,C 180,E1 -16406.576,E2 -16406.576} C_VEL
LIN {X 0,Y 298.42,Z 362.935,A -85,B 0,C 180,E1 -16409.642,E2 -16409.642} C_VEL
LIN {X 0,Y 298.394,Z 362.936,A -85,B 0,C 180,E1 -16412.801,E2 -16412.801} C_VEL
LIN {X 0,Y 298.445,Z 362.931,A -85,B 0,C 180,E1 -16416.808,E2 -16416.808} C_VEL
LIN {X 0,Y 298.386,Z 362.938,A -85,B 0,C 180,E1 -16421.088,E2 -16421.088} C_VEL
LIN {X 0,Y 298.398,Z 362.929,A -85,B 0,C 180,E1 -16423.104,E2 -16423.104} C_VEL
LIN {X 0,Y 298.403,Z 362.94,A -85,B 0,C 180,E1 -16426.922,E2 -16426.922} C_VEL
LIN {X 0,Y 298.399,Z 362.931,A -85,B 0,C 180,E1 -16431.008,E2 -16431.008} C_VEL
LIN {X 0,Y 298.419,Z 362.935,A -85,B 0,C 180,E1 -16433.931,E2 -16433.931} C_VEL
LIN {X 0,Y 298.389,Z 362.936,A -85,B 0,C 180,E1 -16437.986,E2 -16437.986} C_VEL
LIN {X 0,Y 298.424,Z 362.936,A -85,B 0,C 180,E1 -16441.901,E2 -16441.901} C_VEL
LIN {X 0,Y 298.451,Z 362.931,A -85,B 0,C 180,E1 -16444.922,E2 -16444.922} C_VEL
LIN {X 0,Y 298.431,Z 362.929,A -85,B 0,C 180,E1 -16449.315,E2 -16449.315} C_VEL
LIN {X 0,Y 298.451,Z 362.935,A -85,B 0,C 180,E1 -16452.175,E2 -16452.175} C_VEL
LIN {X 0,Y 298.513,Z 362.924,A -85,B 0,C 180,E1 -16454.991,E2 -16454.991} C_VEL
LIN {X 0,Y 298.586,Z 362.915,A -85,B 0,C 180,E1 -16459.147,E2 -16459.147} C_VEL
LIN {X 0,Y 298.701,Z 362.9,A -85,B 0,C 180,E1 -16461.885,E2 -16461.885} C_VEL
LIN {X 0,Y 298.632,Z 362.91,A -85,B 0,C 180,E1 -16464.599,E2 -16464.599} C_VEL
LIN {X 0,Y 298.907,Z 362.879,A -85,B 0,C 180,E1 -16468.653,E2 -16468.653} C_VEL
LIN {X 0,Y 298.842,Z 362.882,A -85,B 0,C 180,E1 -16472.106,E2 -16472.106} C_VEL
LIN {X 0,Y 299.808,Z 365.71,A -85,B 0,C 180,E1 -16472.331,E2 -16472.331} C_VEL
LIN {X 0,Y 311.967,Z 387.524,A -85,B 0,C 180,E1 -16474.462,E2 -16474.462} C_VEL
LIN {X 0,Y 322.521,Z 408.759,A -85,B 0,C 180,E1 -16476.22,E2 -16476.22} C_VEL
LIN {X 0,Y 322.522,Z 412.529,A -85,B 0,C 180,E1 -16476.326,E2 -16476.326} C_VEL
LIN {X 0,Y 318.331,Z 518.965,A -85,B 0,C 180,E1 -16478.891,E2 -16478.891} C_VEL
LIN {X 0,Y 317.277,Z 534.7,A -85,B 0,C 180,E1 -16479.523,E2 -16479.523} C_VEL
LIN {X 0,Y 315.965,Z 549.222,A -85,B 0,C 180,E1 -16480.352,E2 -16480.352} C_VEL
LIN {X 0,Y 314.237,Z 563.519,A -85,B 0,C 180,E1 -16481.417,E2 -16481.417} C_VEL
LIN {X 0,Y 312.108,Z 578.478,A -85,B 0,C 180,E1 -16482.848,E2 -16482.848} C_VEL
LIN {X 0,Y 309.809,Z 591.95,A -85,B 0,C 180,E1 -16484.451,E2 -16484.451} C_VEL
LIN {X 0,Y 307.667,Z 603.691,A -85,B 0,C 180,E1 -16486.155,E2 -16486.155} C_VEL
LIN {X 0,Y 305.535,Z 614.764,A -85,B 0,C 180,E1 -16488.092,E2 -16488.092} C_VEL
LIN {X 0,Y 303.38,Z 625.355,A -85,B 0,C 180,E1 -16490.334,E2 -16490.334} C_VEL
LIN {X 0,Y 301.6,Z 634.24,A -85,B 0,C 180,E1 -16492.613,E2 -16492.613} C_VEL
LIN {X 0,Y 300.079,Z 641.713,A -85,B 0,C 180,E1 -16494.934,E2 -16494.934} C_VEL
LIN {X 0,Y 298.834,Z 648.124,A -85,B 0,C 180,E1 -16497.37,E2 -16497.37} C_VEL
LIN {X 0,Y 298.032,Z 653.047,A -85,B 0,C 180,E1 -16499.684,E2 -16499.684} C_VEL
LIN {X 0,Y 297.469,Z 656.567,A -85,B 0,C 180,E1 -16501.729,E2 -16501.729} C_VEL
LIN {X 0,Y 296.812,Z 660.285,A -85,B 0,C 180,E1 -16504.631,E2 -16504.631} C_VEL
LIN {X 0,Y 296.599,Z 661.828,A -85,B 0,C 180,E1 -16506.327,E2 -16506.327} C_VEL
LIN {X 0,Y 296.483,Z 663.089,A -85,B 0,C 180,E1 -16508.532,E2 -16508.532} C_VEL
LIN {X 0,Y 296.492,Z 663.639,A -85,B 0,C 180,E1 -16510.665,E2 -16510.665} C_VEL
LIN {X 0,Y 296.656,Z 663.273,A -85,B 0,C 180,E1 -16513.396,E2 -16513.396} C_VEL
LIN {X 0,Y 296.919,Z 662.403,A -85,B 0,C 180,E1 -16515.243,E2 -16515.243} C_VEL
LIN {X 0,Y 297.324,Z 660.945,A -85,B 0,C 180,E1 -16517.119,E2 -16517.119} C_VEL
LIN {X 0,Y 298.124,Z 657.919,A -85,B 0,C 180,E1 -16519.771,E2 -16519.771} C_VEL
LIN {X 0,Y 299.441,Z 652.694,A -85,B 0,C 180,E1 -16522.94,E2 -16522.94} C_VEL
LIN {X 0,Y 300.938,Z 647.19,A -85,B 0,C 180,E1 -16525.454,E2 -16525.454} C_VEL
LIN {X 0,Y 302.886,Z 640.047,A -85,B 0,C 180,E1 -16528.042,E2 -16528.042} C_VEL
LIN {X 0,Y 305.162,Z 631.888,A -85,B 0,C 180,E1 -16530.429,E2 -16530.429} C_VEL
LIN {X 0,Y 305.486,Z 628.601,A -85,B 0,C 180,E1 -16531.35,E2 -16531.35} C_VEL
LIN {X 0,Y 304.434,Z 623.175,A -85,B 0,C 180,E1 -16532.9,E2 -16532.9} C_VEL
LIN {X 0,Y 303.494,Z 617.362,A -85,B 0,C 180,E1 -16534.399,E2 -16534.399} C_VEL
LIN {X 0,Y 303.971,Z 613.395,A -85,B 0,C 180,E1 -16535.224,E2 -16535.224} C_VEL
LIN {X 0,Y 306.754,Z 602.467,A -85,B 0,C 180,E1 -16537.077,E2 -16537.077} C_VEL
LIN {X 0,Y 309.683,Z 590.08,A -85,B 0,C 180,E1 -16538.801,E2 -16538.801} C_VEL
LIN {X 0,Y 312.455,Z 576.967,A -85,B 0,C 180,E1 -16540.281,E2 -16540.281} C_VEL
LIN {X 0,Y 314.804,Z 563.279,A -85,B 0,C 180,E1 -16541.539,E2 -16541.539} C_VEL
LIN {X 0,Y 316.806,Z 549.389,A -85,B 0,C 180,E1 -16542.538,E2 -16542.538} C_VEL
LIN {X 0,Y 318.453,Z 534.166,A -85,B 0,C 180,E1 -16543.368,E2 -16543.368} C_VEL
LIN {X 0,Y 319.667,Z 518.708,A -85,B 0,C 180,E1 -16543.943,E2 -16543.943} C_VEL
LIN {X 0,Y 325.071,Z 416.497,A -85,B 0,C 180,E1 -16546.517,E2 -16546.517} C_VEL
LIN {X 0,Y 318.729,Z 404.483,A -85,B 0,C 180,E1 -16548.033,E2 -16548.033} C_VEL
LIN {X 0,Y 311.769,Z 392.928,A -85,B 0,C 180,E1 -16549.79,E2 -16549.79} C_VEL
LIN {X 0,Y 304.909,Z 382.593,A -85,B 0,C 180,E1 -16551.674,E2 -16551.674} C_VEL
LIN {X 0,Y 301.497,Z 377.864,A -85,B 0,C 180,E1 -16552.676,E2 -16552.676} C_VEL
LIN {X 0,Y 298.597,Z 373.765,A -85,B 0,C 180,E1 -16553.581,E2 -16553.581} C_VEL
LIN {X 0,Y 296.089,Z 370.631,A -85,B 0,C 180,E1 -16554.381,E2 -16554.381} C_VEL
LIN {X 0,Y 295.441,Z 369.23,A -85,B 0,C 180,E1 -16554.625,E2 -16554.625} C_VEL
LIN {X 0,Y 293.019,Z 367.334,A -85,B 0,C 180,E1 -16555.399,E2 -16555.399} C_VEL
LIN {X 0,Y 291.823,Z 365.144,A -85,B 0,C 180,E1 -16555.856,E2 -16555.856} C_VEL
LIN {X 0,Y 291.533,Z 363.798,A -85,B 0,C 180,E1 -16556.025,E2 -16556.025} C_VEL
LIN {X 0,Y 291.882,Z 363.752,A -85,B 0,C 180,E1 -16558.62,E2 -16558.62} C_VEL
LIN {X 0,Y 291.887,Z 363.748,A -85,B 0,C 180,E1 -16561.379,E2 -16561.379} C_VEL
LIN {X 0,Y 291.607,Z 363.785,A -85,B 0,C 180,E1 -16565.532,E2 -16565.532} C_VEL
LIN {X 0,Y 291.67,Z 363.779,A -85,B 0,C 180,E1 -16568.909,E2 -16568.909} C_VEL
LIN {X 0,Y 291.519,Z 363.791,A -85,B 0,C 180,E1 -16572.531,E2 -16572.531} C_VEL
LIN {X 0,Y 291.509,Z 363.791,A -85,B 0,C 180,E1 -16575.378,E2 -16575.378} C_VEL
LIN {X 0,Y 291.453,Z 363.805,A -85,B 0,C 180,E1 -16579.874,E2 -16579.874} C_VEL
LIN {X 0,Y 291.403,Z 363.805,A -85,B 0,C 180,E1 -16584.205,E2 -16584.205} C_VEL
LIN {X 0,Y 291.425,Z 363.803,A -85,B 0,C 180,E1 -16587.271,E2 -16587.271} C_VEL
LIN {X 0,Y 291.339,Z 363.816,A -85,B 0,C 180,E1 -16590.436,E2 -16590.436} C_VEL
LIN {X 0,Y 291.346,Z 363.822,A -85,B 0,C 180,E1 -16593.698,E2 -16593.698} C_VEL
LIN {X 0,Y 291.395,Z 363.811,A -85,B 0,C 180,E1 -16597.258,E2 -16597.258} C_VEL
LIN {X 0,Y 291.402,Z 363.984,A -85,B 0,C 180,E1 -16598.407,E2 -16598.407} C_VEL
LIN {X 0,Y 294.116,Z 371.443,A -85,B 0,C 180,E1 -16602.204,E2 -16602.204} C_VEL
LIN {X 0,Y 296.684,Z 378.662,A -85,B 0,C 180,E1 -16605.321,E2 -16605.321} C_VEL
LIN {X 0,Y 299.779,Z 383.739,A -85,B 0,C 180,E1 -16606.338,E2 -16606.338} C_VEL
LIN {X 0,Y 304.704,Z 391.674,A -85,B 0,C 180,E1 -16607.833,E2 -16607.833} C_VEL
LIN {X 0,Y 310.094,Z 401.149,A -85,B 0,C 180,E1 -16609.364,E2 -16609.364} C_VEL
LIN {X 0,Y 316.727,Z 414.467,A -85,B 0,C 180,E1 -16611.14,E2 -16611.14} C_VEL
LIN {X 0,Y 321.529,Z 425.732,A -85,B 0,C 180,E1 -16612.39,E2 -16612.39} C_VEL
LIN {X 0,Y 323.956,Z 445.323,A -85,B 0,C 180,E1 -16613.451,E2 -16613.451} C_VEL
LIN {X 0,Y 318.447,Z 549.876,A -85,B 0,C 180,E1 -16616.085,E2 -16616.085} C_VEL
LIN {X 0,Y 316.755,Z 565.621,A -85,B 0,C 180,E1 -16616.691,E2 -16616.691} C_VEL
LIN {X 0,Y 314.499,Z 581.354,A -85,B 0,C 180,E1 -16617.566,E2 -16617.566} C_VEL
LIN {X 0,Y 311.941,Z 595.504,A -85,B 0,C 180,E1 -16618.6,E2 -16618.6} C_VEL
LIN {X 0,Y 309.454,Z 608.158,A -85,B 0,C 180,E1 -16619.781,E2 -16619.781} C_VEL
LIN {X 0,Y 306.281,Z 622.025,A -85,B 0,C 180,E1 -16621.379,E2 -16621.379} C_VEL
LIN {X 0,Y 303.169,Z 634.356,A -85,B 0,C 180,E1 -16623.124,E2 -16623.124} C_VEL
LIN {X 0,Y 300.214,Z 645.705,A -85,B 0,C 180,E1 -16625.078,E2 -16625.078} C_VEL
LIN {X 0,Y 297.215,Z 657.152,A -85,B 0,C 180,E1 -16627.496,E2 -16627.496} C_VEL
LIN {X 0,Y 294.928,Z 666.065,A -85,B 0,C 180,E1 -16629.785,E2 -16629.785} C_VEL
LIN {X 0,Y 292.733,Z 674.823,A -85,B 0,C 180,E1 -16632.536,E2 -16632.536} C_VEL
LIN {X 0,Y 291.196,Z 681.967,A -85,B 0,C 180,E1 -16635.338,E2 -16635.338} C_VEL
LIN {X 0,Y 290.194,Z 687.553,A -85,B 0,C 180,E1 -16638.12,E2 -16638.12} C_VEL
LIN {X 0,Y 289.751,Z 690.862,A -85,B 0,C 180,E1 -16640.224,E2 -16640.224} C_VEL
LIN {X 0,Y 289.552,Z 694.218,A -85,B 0,C 180,E1 -16643.029,E2 -16643.029} C_VEL
LIN {X 0,Y 289.554,Z 696.338,A -85,B 0,C 180,E1 -16645.824,E2 -16645.824} C_VEL
LIN {X 0,Y 289.64,Z 697.218,A -85,B 0,C 180,E1 -16648.609,E2 -16648.609} C_VEL
LIN {X 0,Y 289.757,Z 697.216,A -85,B 0,C 180,E1 -16649.999,E2 -16649.999} C_VEL
LIN {X 0,Y 289.599,Z 696.281,A -85,B 0,C 180,E1 -16652.781,E2 -16652.781} C_VEL
LIN {X 0,Y 289.584,Z 693.978,A -85,B 0,C 180,E1 -16655.712,E2 -16655.712} C_VEL
LIN {X 0,Y 289.671,Z 690.692,A -85,B 0,C 180,E1 -16658.37,E2 -16658.37} C_VEL
LIN {X 0,Y 289.98,Z 685.891,A -85,B 0,C 180,E1 -16661.179,E2 -16661.179} C_VEL
LIN {X 0,Y 290.819,Z 679.609,A -85,B 0,C 180,E1 -16663.984,E2 -16663.984} C_VEL
LIN {X 0,Y 292.144,Z 671.667,A -85,B 0,C 180,E1 -16666.778,E2 -16666.778} C_VEL
LIN {X 0,Y 293.707,Z 663.181,A -85,B 0,C 180,E1 -16669.209,E2 -16669.209} C_VEL
LIN {X 0,Y 295.848,Z 652.946,A -85,B 0,C 180,E1 -16671.604,E2 -16671.604} C_VEL
LIN {X 0,Y 297.896,Z 642.45,A -85,B 0,C 180,E1 -16673.644,E2 -16673.644} C_VEL
LIN {X 0,Y 300.225,Z 631.045,A -85,B 0,C 180,E1 -16675.476,E2 -16675.476} C_VEL
LIN {X 0,Y 302.607,Z 618.691,A -85,B 0,C 180,E1 -16677.115,E2 -16677.115} C_VEL
LIN {X 0,Y 305,Z 605.284,A -85,B 0,C 180,E1 -16678.563,E2 -16678.563} C_VEL
LIN {X 0,Y 307.276,Z 590.187,A -85,B 0,C 180,E1 -16679.864,E2 -16679.864} C_VEL
LIN {X 0,Y 309.216,Z 575.099,A -85,B 0,C 180,E1 -16680.85,E2 -16680.85} C_VEL
LIN {X 0,Y 310.777,Z 559.674,A -85,B 0,C 180,E1 -16681.577,E2 -16681.577} C_VEL
LIN {X 0,Y 311.778,Z 543.415,A -85,B 0,C 180,E1 -16682.082,E2 -16682.082} C_VEL
LIN {X 0,Y 315.76,Z 443.617,A -85,B 0,C 180,E1 -16684.511,E2 -16684.511} C_VEL
LIN {X 0,Y 311.565,Z 416.621,A -85,B 0,C 180,E1 -16685.75,E2 -16685.75} C_VEL
LIN {X 0,Y 302.863,Z 396.546,A -85,B 0,C 180,E1 -16687.366,E2 -16687.366} C_VEL
LIN {X 0,Y 296.969,Z 383.956,A -85,B 0,C 180,E1 -16688.533,E2 -16688.533} C_VEL
LIN {X 0,Y 293.969,Z 372.956,A -85,B 0,C 180,E1 -16691.661,E2 -16691.661} C_VEL
LIN {X 0,Y 291.339,Z 363.817,A -85,B 0,C 180,E1 -16694.451,E2 -16694.451} C_VEL
LIN {X 0,Y 291.323,Z 363.814,A -85,B 0,C 180,E1 -16698.404,E2 -16698.404} C_VEL
LIN {X 0,Y 291.349,Z 363.814,A -85,B 0,C 180,E1 -16701.158,E2 -16701.158} C_VEL
LIN {X 0,Y 291.358,Z 363.82,A -85,B 0,C 180,E1 -16704.626,E2 -16704.626} C_VEL
LIN {X 0,Y 291.368,Z 363.815,A -85,B 0,C 180,E1 -16707.951,E2 -16707.951} C_VEL
LIN {X 0,Y 291.379,Z 363.816,A -85,B 0,C 180,E1 -16711.158,E2 -16711.158} C_VEL
LIN {X 0,Y 291.413,Z 363.806,A -85,B 0,C 180,E1 -16714.272,E2 -16714.272} C_VEL
LIN {X 0,Y 291.378,Z 363.813,A -85,B 0,C 180,E1 -16717.3,E2 -16717.3} C_VEL
LIN {X 0,Y 291.454,Z 363.804,A -85,B 0,C 180,E1 -16720.27,E2 -16720.27} C_VEL
LIN {X 0,Y 291.552,Z 363.794,A -85,B 0,C 180,E1 -16724.624,E2 -16724.624} C_VEL
LIN {X 0,Y 291.533,Z 363.778,A -85,B 0,C 180,E1 -16728.881,E2 -16728.881} C_VEL
LIN {X 0,Y 291.703,Z 363.768,A -85,B 0,C 180,E1 -16731.689,E2 -16731.689} C_VEL
LIN {X 0,Y 291.626,Z 363.783,A -85,B 0,C 180,E1 -16734.469,E2 -16734.469} C_VEL
LIN {X 0,Y 291.887,Z 363.741,A -85,B 0,C 180,E1 -16738.621,E2 -16738.621} C_VEL
LIN {X 0,Y 291.887,Z 363.75,A -85,B 0,C 180,E1 -16741.38,E2 -16741.38} C_VEL
LIN {X 0,Y 291.744,Z 363.758,A -85,B 0,C 180,E1 -16746.918,E2 -16746.918} C_VEL
LIN {X 0,Y 291.627,Z 363.779,A -85,B 0,C 180,E1 -16749.712,E2 -16749.712} C_VEL
LIN {X 0,Y 291.52,Z 363.792,A -85,B 0,C 180,E1 -16753.951,E2 -16753.951} C_VEL
LIN {X 0,Y 291.485,Z 363.79,A -85,B 0,C 180,E1 -16756.819,E2 -16756.819} C_VEL
LIN {X 0,Y 291.449,Z 363.802,A -85,B 0,C 180,E1 -16759.876,E2 -16759.876} C_VEL
LIN {X 0,Y 291.381,Z 363.809,A -85,B 0,C 180,E1 -16764.208,E2 -16764.208} C_VEL
LIN {X 0,Y 291.419,Z 363.803,A -85,B 0,C 180,E1 -16767.272,E2 -16767.272} C_VEL
LIN {X 0,Y 291.336,Z 363.82,A -85,B 0,C 180,E1 -16770.438,E2 -16770.438} C_VEL
LIN {X 0,Y 291.344,Z 363.81,A -85,B 0,C 180,E1 -16773.699,E2 -16773.699} C_VEL
LIN {X 0,Y 291.375,Z 363.812,A -85,B 0,C 180,E1 -16777.255,E2 -16777.255} C_VEL
LIN {X 0,Y 291.332,Z 363.82,A -85,B 0,C 180,E1 -16780.643,E2 -16780.643} C_VEL
LIN {X 0,Y 291.289,Z 363.816,A -85,B 0,C 180,E1 -16784.403,E2 -16784.403} C_VEL
LIN {X 0,Y 291.326,Z 363.823,A -85,B 0,C 180,E1 -16788.405,E2 -16788.405} C_VEL
LIN {X 0,Y 291.348,Z 363.809,A -85,B 0,C 180,E1 -16791.158,E2 -16791.158} C_VEL
LIN {X 0,Y 291.362,Z 363.819,A -85,B 0,C 180,E1 -16794.627,E2 -16794.627} C_VEL
LIN {X 0,Y 291.367,Z 363.81,A -85,B 0,C 180,E1 -16797.951,E2 -16797.951} C_VEL
LIN {X 0,Y 291.353,Z 363.817,A -85,B 0,C 180,E1 -16801.156,E2 -16801.156} C_VEL
LIN {X 0,Y 291.377,Z 363.81,A -85,B 0,C 180,E1 -16804.269,E2 -16804.269} C_VEL
LIN {X 0,Y 291.377,Z 363.813,A -85,B 0,C 180,E1 -16807.3,E2 -16807.3} C_VEL
LIN {X 0,Y 291.408,Z 363.807,A -85,B 0,C 180,E1 -16810.267,E2 -16810.267} C_VEL
LIN {X 0,Y 291.476,Z 363.8,A -85,B 0,C 180,E1 -16814.683,E2 -16814.683} C_VEL
LIN {X 0,Y 291.531,Z 363.795,A -85,B 0,C 180,E1 -16818.881,E2 -16818.881} C_VEL
LIN {X 0,Y 291.655,Z 363.777,A -85,B 0,C 180,E1 -16821.688,E2 -16821.688} C_VEL
LIN {X 0,Y 291.602,Z 363.785,A -85,B 0,C 180,E1 -16824.468,E2 -16824.468} C_VEL
LIN {X 0,Y 291.874,Z 363.755,A -85,B 0,C 180,E1 -16828.621,E2 -16828.621} C_VEL
LIN {X 0,Y 291.857,Z 363.755,A -85,B 0,C 180,E1 -16831.208,E2 -16831.208} C_VEL
LIN {X 0,Y 292.998,Z 366.823,A -85,B 0,C 180,E1 -16831.484,E2 -16831.484} C_VEL
LIN {X 0,Y 298.007,Z 375.866,A -85,B 0,C 180,E1 -16832.425,E2 -16832.425} C_VEL
LIN {X 0,Y 306.708,Z 391.441,A -85,B 0,C 180,E1 -16833.968,E2 -16833.968} C_VEL
LIN {X 0,Y 316.487,Z 411.181,A -85,B 0,C 180,E1 -16835.654,E2 -16835.654} C_VEL
LIN {X 0,Y 311.991,Z 519.612,A -85,B 0,C 180,E1 -16838.315,E2 -16838.315} C_VEL
LIN {X 0,Y 310.931,Z 535.212,A -85,B 0,C 180,E1 -16838.959,E2 -16838.959} C_VEL
LIN {X 0,Y 309.568,Z 549.725,A -85,B 0,C 180,E1 -16839.804,E2 -16839.804} C_VEL
LIN {X 0,Y 307.759,Z 564.137,A -85,B 0,C 180,E1 -16840.899,E2 -16840.899} C_VEL
LIN {X 0,Y 305.679,Z 578.361,A -85,B 0,C 180,E1 -16842.279,E2 -16842.279} C_VEL
LIN {X 0,Y 303.487,Z 590.982,A -85,B 0,C 180,E1 -16843.782,E2 -16843.782} C_VEL
LIN {X 0,Y 301.185,Z 603.245,A -85,B 0,C 180,E1 -16845.566,E2 -16845.566} C_VEL
LIN {X 0,Y 299.072,Z 613.876,A -85,B 0,C 180,E1 -16847.435,E2 -16847.435} C_VEL
LIN {X 0,Y 296.767,Z 624.728,A -85,B 0,C 180,E1 -16849.723,E2 -16849.723} C_VEL
LIN {X 0,Y 294.885,Z 633.675,A -85,B 0,C 180,E1 -16852.024,E2 -16852.024} C_VEL
LIN {X 0,Y 293.287,Z 641.349,A -85,B 0,C 180,E1 -16854.411,E2 -16854.411} C_VEL
LIN {X 0,Y 291.817,Z 648.7,A -85,B 0,C 180,E1 -16857.232,E2 -16857.232} C_VEL
LIN {X 0,Y 290.983,Z 653.584,A -85,B 0,C 180,E1 -16859.599,E2 -16859.599} C_VEL
LIN {X 0,Y 290.272,Z 657.794,A -85,B 0,C 180,E1 -16862.186,E2 -16862.186} C_VEL
LIN {X 0,Y 289.762,Z 660.536,A -85,B 0,C 180,E1 -16864.446,E2 -16864.446} C_VEL
LIN {X 0,Y 289.418,Z 662.907,A -85,B 0,C 180,E1 -16867.379,E2 -16867.379} C_VEL
LIN {X 0,Y 289.375,Z 663.725,A -85,B 0,C 180,E1 -16869.158,E2 -16869.158} C_VEL
LIN {X 0,Y 289.412,Z 664.088,A -85,B 0,C 180,E1 -16871.166,E2 -16871.166} C_VEL
LIN {X 0,Y 289.552,Z 663.786,A -85,B 0,C 180,E1 -16873.267,E2 -16873.267} C_VEL
LIN {X 0,Y 289.866,Z 662.903,A -85,B 0,C 180,E1 -16875.321,E2 -16875.321} C_VEL
LIN {X 0,Y 290.314,Z 661.432,A -85,B 0,C 180,E1 -16877.325,E2 -16877.325} C_VEL
LIN {X 0,Y 290.898,Z 659.351,A -85,B 0,C 180,E1 -16879.283,E2 -16879.283} C_VEL
LIN {X 0,Y 291.873,Z 655.63,A -85,B 0,C 180,E1 -16881.924,E2 -16881.924} C_VEL
LIN {X 0,Y 293.493,Z 649.897,A -85,B 0,C 180,E1 -16884.92,E2 -16884.92} C_VEL
LIN {X 0,Y 295.5,Z 643.128,A -85,B 0,C 180,E1 -16887.647,E2 -16887.647} C_VEL
LIN {X 0,Y 297.528,Z 636.267,A -85,B 0,C 180,E1 -16889.891,E2 -16889.891} C_VEL
LIN {X 0,Y 300.349,Z 626.712,A -85,B 0,C 180,E1 -16892.427,E2 -16892.427} C_VEL
LIN {X 0,Y 303.245,Z 616.31,A -85,B 0,C 180,E1 -16894.672,E2 -16894.672} C_VEL
LIN {X 0,Y 303.971,Z 613.395,A -85,B 0,C 180,E1 -16895.224,E2 -16895.224} C_VEL
LIN {X 0,Y 304.483,Z 609.351,A -85,B 0,C 180,E1 -16896.03,E2 -16896.03} C_VEL
LIN {X 0,Y 303.762,Z 602.797,A -85,B 0,C 180,E1 -16897.428,E2 -16897.428} C_VEL
LIN {X 0,Y 303.078,Z 595.888,A -85,B 0,C 180,E1 -16898.758,E2 -16898.758} C_VEL
LIN {X 0,Y 303.613,Z 591.278,A -85,B 0,C 180,E1 -16899.444,E2 -16899.444} C_VEL
LIN {X 0,Y 306.402,Z 578.676,A -85,B 0,C 180,E1 -16900.913,E2 -16900.913} C_VEL
LIN {X 0,Y 309.007,Z 564.558,A -85,B 0,C 180,E1 -16902.249,E2 -16902.249} C_VEL
LIN {X 0,Y 311.074,Z 551.065,A -85,B 0,C 180,E1 -16903.258,E2 -16903.258} C_VEL
LIN {X 0,Y 312.86,Z 536.03,A -85,B 0,C 180,E1 -16904.11,E2 -16904.11} C_VEL
LIN {X 0,Y 314.138,Z 521.122,A -85,B 0,C 180,E1 -16904.701,E2 -16904.701} C_VEL
LIN {X 0,Y 319.731,Z 419.071,A -85,B 0,C 180,E1 -16907.327,E2 -16907.327} C_VEL
LIN {X 0,Y 313.965,Z 408.252,A -85,B 0,C 180,E1 -16908.776,E2 -16908.776} C_VEL
LIN {X 0,Y 308.105,Z 398.221,A -85,B 0,C 180,E1 -16910.336,E2 -16910.336} C_VEL
LIN {X 0,Y 301.265,Z 387.841,A -85,B 0,C 180,E1 -16912.291,E2 -16912.291} C_VEL
LIN {X 0,Y 298.047,Z 383.254,A -85,B 0,C 180,E1 -16913.282,E2 -16913.282} C_VEL
LIN {X 0,Y 295.256,Z 379.332,A -85,B 0,C 180,E1 -16914.187,E2 -16914.187} C_VEL
LIN {X 0,Y 292.74,Z 375.871,A -85,B 0,C 180,E1 -16915.05,E2 -16915.05} C_VEL
LIN {X 0,Y 289.596,Z 372.421,A -85,B 0,C 180,E1 -16916.136,E2 -16916.136} C_VEL
LIN {X 0,Y 288.24,Z 370.009,A -85,B 0,C 180,E1 -16916.68,E2 -16916.68} C_VEL
LIN {X 0,Y 285.957,Z 367.819,A -85,B 0,C 180,E1 -16917.534,E2 -16917.534} C_VEL
LIN {X 0,Y 284.92,Z 365.478,A -85,B 0,C 180,E1 -16918.012,E2 -16918.012} C_VEL
LIN {X 0,Y 284.786,Z 364.637,A -85,B 0,C 180,E1 -16918.143,E2 -16918.143} C_VEL
LIN {X 0,Y 284.853,Z 364.624,A -85,B 0,C 180,E1 -16921.413,E2 -16921.413} C_VEL
LIN {X 0,Y 284.646,Z 364.647,A -85,B 0,C 180,E1 -16927.091,E2 -16927.091} C_VEL
LIN {X 0,Y 284.517,Z 364.662,A -85,B 0,C 180,E1 -16929.957,E2 -16929.957} C_VEL
LIN {X 0,Y 284.466,Z 364.676,A -85,B 0,C 180,E1 -16934.303,E2 -16934.303} C_VEL
LIN {X 0,Y 284.388,Z 364.677,A -85,B 0,C 180,E1 -16938.739,E2 -16938.739} C_VEL
LIN {X 0,Y 284.369,Z 364.687,A -85,B 0,C 180,E1 -16943.292,E2 -16943.292} C_VEL
LIN {X 0,Y 284.399,Z 364.678,A -85,B 0,C 180,E1 -16947.173,E2 -16947.173} C_VEL
LIN {X 0,Y 284.298,Z 364.699,A -85,B 0,C 180,E1 -16951.274,E2 -16951.274} C_VEL
LIN {X 0,Y 284.363,Z 364.687,A -85,B 0,C 180,E1 -16955.353,E2 -16955.353} C_VEL
LIN {X 0,Y 284.347,Z 364.707,A -85,B 0,C 180,E1 -16956.238,E2 -16956.238} C_VEL
LIN {X 0,Y 286.462,Z 370.555,A -85,B 0,C 180,E1 -16959.633,E2 -16959.633} C_VEL
LIN {X 0,Y 289.021,Z 377.609,A -85,B 0,C 180,E1 -16963.126,E2 -16963.126} C_VEL
LIN {X 0,Y 292.359,Z 382.822,A -85,B 0,C 180,E1 -16964.356,E2 -16964.356} C_VEL
LIN {X 0,Y 293.79,Z 384.988,A -85,B 0,C 180,E1 -16964.859,E2 -16964.859} C_VEL
LIN {X 0,Y 298.195,Z 392.086,A -85,B 0,C 180,E1 -16966.324,E2 -16966.324} C_VEL
LIN {X 0,Y 301.455,Z 397.58,A -85,B 0,C 180,E1 -16967.344,E2 -16967.344} C_VEL
LIN {X 0,Y 306.314,Z 406.338,A -85,B 0,C 180,E1 -16968.785,E2 -16968.785} C_VEL
LIN {X 0,Y 312.424,Z 418.867,A -85,B 0,C 180,E1 -16970.502,E2 -16970.502} C_VEL
LIN {X 0,Y 316.577,Z 428.641,A -85,B 0,C 180,E1 -16971.629,E2 -16971.629} C_VEL
LIN {X 0,Y 318.683,Z 446.856,A -85,B 0,C 180,E1 -16972.641,E2 -16972.641} C_VEL
LIN {X 0,Y 313.05,Z 548.365,A -85,B 0,C 180,E1 -16975.223,E2 -16975.223} C_VEL
LIN {X 0,Y 311.327,Z 564.367,A -85,B 0,C 180,E1 -16975.837,E2 -16975.837} C_VEL
LIN {X 0,Y 308.966,Z 580.223,A -85,B 0,C 180,E1 -16976.717,E2 -16976.717} C_VEL
LIN {X 0,Y 306.339,Z 594.493,A -85,B 0,C 180,E1 -16977.764,E2 -16977.764} C_VEL
LIN {X 0,Y 303.476,Z 608.104,A -85,B 0,C 180,E1 -16979.041,E2 -16979.041} C_VEL
LIN {X 0,Y 300.368,Z 621.197,A -85,B 0,C 180,E1 -16980.57,E2 -16980.57} C_VEL
LIN {X 0,Y 296.857,Z 634.581,A -85,B 0,C 180,E1 -16982.505,E2 -16982.505} C_VEL
LIN {X 0,Y 293.759,Z 645.8,A -85,B 0,C 180,E1 -16984.491,E2 -16984.491} C_VEL
LIN {X 0,Y 290.791,Z 656.621,A -85,B 0,C 180,E1 -16986.836,E2 -16986.836} C_VEL
LIN {X 0,Y 288.229,Z 665.982,A -85,B 0,C 180,E1 -16989.294,E2 -16989.294} C_VEL
LIN {X 0,Y 285.881,Z 674.667,A -85,B 0,C 180,E1 -16992.103,E2 -16992.103} C_VEL
LIN {X 0,Y 284.21,Z 681.946,A -85,B 0,C 180,E1 -16995.068,E2 -16995.068} C_VEL
LIN {X 0,Y 283.187,Z 687.286,A -85,B 0,C 180,E1 -16997.821,E2 -16997.821} C_VEL
LIN {X 0,Y 282.698,Z 690.558,A -85,B 0,C 180,E1 -16999.978,E2 -16999.978} C_VEL
LIN {X 0,Y 282.465,Z 693.871,A -85,B 0,C 180,E1 -17002.853,E2 -17002.853} C_VEL
LIN {X 0,Y 282.472,Z 695.967,A -85,B 0,C 180,E1 -17005.719,E2 -17005.719} C_VEL
LIN {X 0,Y 282.55,Z 696.814,A -85,B 0,C 180,E1 -17008.574,E2 -17008.574} C_VEL
LIN {X 0,Y 282.668,Z 696.79,A -85,B 0,C 180,E1 -17009.999,E2 -17009.999} C_VEL
LIN {X 0,Y 282.522,Z 695.814,A -85,B 0,C 180,E1 -17012.851,E2 -17012.851} C_VEL
LIN {X 0,Y 282.505,Z 693.615,A -85,B 0,C 180,E1 -17015.71,E2 -17015.71} C_VEL
LIN {X 0,Y 282.593,Z 690.13,A -85,B 0,C 180,E1 -17018.581,E2 -17018.581} C_VEL
LIN {X 0,Y 282.947,Z 685.274,A -85,B 0,C 180,E1 -17021.461,E2 -17021.461} C_VEL
LIN {X 0,Y 283.832,Z 678.928,A -85,B 0,C 180,E1 -17024.336,E2 -17024.336} C_VEL
LIN {X 0,Y 285.221,Z 670.909,A -85,B 0,C 180,E1 -17027.198,E2 -17027.198} C_VEL
LIN {X 0,Y 286.917,Z 662.345,A -85,B 0,C 180,E1 -17029.682,E2 -17029.682} C_VEL
LIN {X 0,Y 288.79,Z 653.699,A -85,B 0,C 180,E1 -17031.765,E2 -17031.765} C_VEL
LIN {X 0,Y 290.884,Z 643.287,A -85,B 0,C 180,E1 -17033.871,E2 -17033.871} C_VEL
LIN {X 0,Y 293.2,Z 632.103,A -85,B 0,C 180,E1 -17035.75,E2 -17035.75} C_VEL
LIN {X 0,Y 295.62,Z 620.044,A -85,B 0,C 180,E1 -17037.426,E2 -17037.426} C_VEL
LIN {X 0,Y 298.113,Z 607.031,A -85,B 0,C 180,E1 -17038.899,E2 -17038.899} C_VEL
LIN {X 0,Y 300.37,Z 593.209,A -85,B 0,C 180,E1 -17040.163,E2 -17040.163} C_VEL
LIN {X 0,Y 302.308,Z 579.479,A -85,B 0,C 180,E1 -17041.148,E2 -17041.148} C_VEL
LIN {X 0,Y 303.949,Z 565.013,A -85,B 0,C 180,E1 -17041.932,E2 -17041.932} C_VEL
LIN {X 0,Y 305.171,Z 549.413,A -85,B 0,C 180,E1 -17042.52,E2 -17042.52} C_VEL
LIN {X 0,Y 309.617,Z 445.907,A -85,B 0,C 180,E1 -17045.097,E2 -17045.097} C_VEL
LIN {X 0,Y 306.797,Z 425.633,A -85,B 0,C 180,E1 -17046.016,E2 -17046.016} C_VEL
LIN {X 0,Y 305.603,Z 418.981,A -85,B 0,C 180,E1 -17046.354,E2 -17046.354} C_VEL
LIN {X 0,Y 297.342,Z 399.939,A -85,B 0,C 180,E1 -17047.935,E2 -17047.935} C_VEL
LIN {X 0,Y 289.606,Z 383.479,A -85,B 0,C 180,E1 -17049.515,E2 -17049.515} C_VEL
LIN {X 0,Y 286.647,Z 372.871,A -85,B 0,C 180,E1 -17052.648,E2 -17052.648} C_VEL
LIN {X 0,Y 284.283,Z 364.695,A -85,B 0,C 180,E1 -17055.229,E2 -17055.229} C_VEL
LIN {X 0,Y 284.268,Z 364.692,A -85,B 0,C 180,E1 -17058.124,E2 -17058.124} C_VEL
LIN {X 0,Y 284.319,Z 364.689,A -85,B 0,C 180,E1 -17062.278,E2 -17062.278} C_VEL
LIN {X 0,Y 284.305,Z 364.694,A -85,B 0,C 180,E1 -17065.351,E2 -17065.351} C_VEL
LIN {X 0,Y 284.292,Z 364.698,A -85,B 0,C 180,E1 -17068.726,E2 -17068.726} C_VEL
LIN {X 0,Y 284.394,Z 364.687,A -85,B 0,C 180,E1 -17072.826,E2 -17072.826} C_VEL
LIN {X 0,Y 284.363,Z 364.689,A -85,B 0,C 180,E1 -17076.707,E2 -17076.707} C_VEL
LIN {X 0,Y 284.4,Z 364.682,A -85,B 0,C 180,E1 -17081.262,E2 -17081.262} C_VEL
LIN {X 0,Y 284.489,Z 364.673,A -85,B 0,C 180,E1 -17084.459,E2 -17084.459} C_VEL
LIN {X 0,Y 284.485,Z 364.655,A -85,B 0,C 180,E1 -17088.602,E2 -17088.602} C_VEL
LIN {X 0,Y 284.654,Z 364.647,A -85,B 0,C 180,E1 -17091.481,E2 -17091.481} C_VEL
LIN {X 0,Y 284.596,Z 364.658,A -85,B 0,C 180,E1 -17094.332,E2 -17094.332} C_VEL
LIN {X 0,Y 284.853,Z 364.616,A -85,B 0,C 180,E1 -17098.587,E2 -17098.587} C_VEL
LIN {X 0,Y 284.853,Z 364.626,A -85,B 0,C 180,E1 -17101.414,E2 -17101.414} C_VEL
LIN {X 0,Y 284.696,Z 364.635,A -85,B 0,C 180,E1 -17107.091,E2 -17107.091} C_VEL
LIN {X 0,Y 284.564,Z 364.659,A -85,B 0,C 180,E1 -17109.956,E2 -17109.956} C_VEL
LIN {X 0,Y 284.48,Z 364.67,A -85,B 0,C 180,E1 -17114.303,E2 -17114.303} C_VEL
LIN {X 0,Y 284.424,Z 364.671,A -85,B 0,C 180,E1 -17117.249,E2 -17117.249} C_VEL
LIN {X 0,Y 284.376,Z 364.685,A -85,B 0,C 180,E1 -17120.243,E2 -17120.243} C_VEL
LIN {X 0,Y 284.335,Z 364.679,A -85,B 0,C 180,E1 -17124.848,E2 -17124.848} C_VEL
LIN {X 0,Y 284.329,Z 364.686,A -85,B 0,C 180,E1 -17128.012,E2 -17128.012} C_VEL
LIN {X 0,Y 284.295,Z 364.695,A -85,B 0,C 180,E1 -17131.275,E2 -17131.275} C_VEL
LIN {X 0,Y 284.34,Z 364.68,A -85,B 0,C 180,E1 -17135.349,E2 -17135.349} C_VEL
LIN {X 0,Y 284.311,Z 364.692,A -85,B 0,C 180,E1 -17138.17,E2 -17138.17} C_VEL
LIN {X 0,Y 284.269,Z 364.696,A -85,B 0,C 180,E1 -17142.125,E2 -17142.125} C_VEL
LIN {X 0,Y 284.255,Z 364.699,A -85,B 0,C 180,E1 -17146.19,E2 -17146.19} C_VEL
LIN {X 0,Y 284.307,Z 364.692,A -85,B 0,C 180,E1 -17150.025,E2 -17150.025} C_VEL
LIN {X 0,Y 284.331,Z 364.69,A -85,B 0,C 180,E1 -17153.615,E2 -17153.615} C_VEL
LIN {X 0,Y 284.307,Z 364.689,A -85,B 0,C 180,E1 -17157.191,E2 -17157.191} C_VEL
LIN {X 0,Y 284.342,Z 364.69,A -85,B 0,C 180,E1 -17160.375,E2 -17160.375} C_VEL
LIN {X 0,Y 284.315,Z 364.689,A -85,B 0,C 180,E1 -17163.581,E2 -17163.581} C_VEL
LIN {X 0,Y 284.334,Z 364.693,A -85,B 0,C 180,E1 -17166.705,E2 -17166.705} C_VEL
LIN {X 0,Y 284.379,Z 364.68,A -85,B 0,C 180,E1 -17169.905,E2 -17169.905} C_VEL
LIN {X 0,Y 284.417,Z 364.679,A -85,B 0,C 180,E1 -17174.517,E2 -17174.517} C_VEL
LIN {X 0,Y 284.467,Z 364.673,A -85,B 0,C 180,E1 -17178.601,E2 -17178.601} C_VEL
LIN {X 0,Y 284.612,Z 364.654,A -85,B 0,C 180,E1 -17181.48,E2 -17181.48} C_VEL
LIN {X 0,Y 284.572,Z 364.662,A -85,B 0,C 180,E1 -17184.331,E2 -17184.331} C_VEL
LIN {X 0,Y 284.841,Z 364.631,A -85,B 0,C 180,E1 -17188.587,E2 -17188.587} C_VEL
LIN {X 0,Y 284.826,Z 364.629,A -85,B 0,C 180,E1 -17190.265,E2 -17190.265} C_VEL
LIN {X 0,Y 285.893,Z 367.612,A -85,B 0,C 180,E1 -17190.545,E2 -17190.545} C_VEL
LIN {X 0,Y 287.295,Z 369.722,A -85,B 0,C 180,E1 -17190.809,E2 -17190.809} C_VEL
LIN {X 0,Y 302.001,Z 396.414,A -85,B 0,C 180,E1 -17193.562,E2 -17193.562} C_VEL
LIN {X 0,Y 310.201,Z 413.206,A -85,B 0,C 180,E1 -17195.021,E2 -17195.021} C_VEL
LIN {X 0,Y 305.747,Z 519.724,A -85,B 0,C 180,E1 -17197.699,E2 -17197.699} C_VEL
LIN {X 0,Y 304.63,Z 535.383,A -85,B 0,C 180,E1 -17198.352,E2 -17198.352} C_VEL
LIN {X 0,Y 303.143,Z 550.468,A -85,B 0,C 180,E1 -17199.248,E2 -17199.248} C_VEL
LIN {X 0,Y 301.194,Z 565.409,A -85,B 0,C 180,E1 -17200.419,E2 -17200.419} C_VEL
LIN {X 0,Y 299.271,Z 578.231,A -85,B 0,C 180,E1 -17201.686,E2 -17201.686} C_VEL
LIN {X 0,Y 296.925,Z 591.401,A -85,B 0,C 180,E1 -17203.282,E2 -17203.282} C_VEL
LIN {X 0,Y 294.374,Z 604.406,A -85,B 0,C 180,E1 -17205.226,E2 -17205.226} C_VEL
LIN {X 0,Y 292.214,Z 614.96,A -85,B 0,C 180,E1 -17207.136,E2 -17207.136} C_VEL
LIN {X 0,Y 289.881,Z 625.563,A -85,B 0,C 180,E1 -17209.445,E2 -17209.445} C_VEL
LIN {X 0,Y 287.852,Z 634.828,A -85,B 0,C 180,E1 -17211.907,E2 -17211.907} C_VEL
LIN {X 0,Y 285.999,Z 643.337,A -85,B 0,C 180,E1 -17214.693,E2 -17214.693} C_VEL
LIN {X 0,Y 284.69,Z 649.719,A -85,B 0,C 180,E1 -17217.286,E2 -17217.286} C_VEL
LIN {X 0,Y 283.78,Z 654.822,A -85,B 0,C 180,E1 -17219.91,E2 -17219.91} C_VEL
LIN {X 0,Y 283.106,Z 658.636,A -85,B 0,C 180,E1 -17222.43,E2 -17222.43} C_VEL
LIN {X 0,Y 282.612,Z 661.445,A -85,B 0,C 180,E1 -17224.888,E2 -17224.888} C_VEL
LIN {X 0,Y 282.348,Z 663.191,A -85,B 0,C 180,E1 -17227.2,E2 -17227.2} C_VEL
LIN {X 0,Y 282.298,Z 664.388,A -85,B 0,C 180,E1 -17230.338,E2 -17230.338} C_VEL
LIN {X 0,Y 282.372,Z 664.448,A -85,B 0,C 180,E1 -17232.223,E2 -17232.223} C_VEL
LIN {X 0,Y 282.572,Z 664.012,A -85,B 0,C 180,E1 -17234.14,E2 -17234.14} C_VEL
LIN {X 0,Y 282.924,Z 663.011,A -85,B 0,C 180,E1 -17236.087,E2 -17236.087} C_VEL
LIN {X 0,Y 283.729,Z 660.495,A -85,B 0,C 180,E1 -17239.015,E2 -17239.015} C_VEL
LIN {X 0,Y 284.894,Z 656.391,A -85,B 0,C 180,E1 -17242.131,E2 -17242.131} C_VEL
LIN {X 0,Y 286.473,Z 651.268,A -85,B 0,C 180,E1 -17244.958,E2 -17244.958} C_VEL
LIN {X 0,Y 288.745,Z 643.976,A -85,B 0,C 180,E1 -17248.03,E2 -17248.03} C_VEL
LIN {X 0,Y 291.335,Z 635.548,A -85,B 0,C 180,E1 -17250.806,E2 -17250.806} C_VEL
LIN {X 0,Y 293.897,Z 627.477,A -85,B 0,C 180,E1 -17252.976,E2 -17252.976} C_VEL
LIN {X 0,Y 297.045,Z 616.727,A -85,B 0,C 180,E1 -17255.354,E2 -17255.354} C_VEL
LIN {X 0,Y 300.185,Z 605.051,A -85,B 0,C 180,E1 -17257.457,E2 -17257.457} C_VEL
LIN {X 0,Y 303.068,Z 593.608,A -85,B 0,C 180,E1 -17259.147,E2 -17259.147} C_VEL
LIN {X 0,Y 303.613,Z 591.278,A -85,B 0,C 180,E1 -17259.444,E2 -17259.444} C_VEL
LIN {X 0,Y 304.167,Z 586.577,A -85,B 0,C 180,E1 -17260.109,E2 -17260.109} C_VEL
LIN {X 0,Y 303.573,Z 578.981,A -85,B 0,C 180,E1 -17261.314,E2 -17261.314} C_VEL
LIN {X 0,Y 302.888,Z 571.131,A -85,B 0,C 180,E1 -17262.447,E2 -17262.447} C_VEL
LIN {X 0,Y 303.262,Z 565.985,A -85,B 0,C 180,E1 -17262.987,E2 -17262.987} C_VEL
LIN {X 0,Y 305.527,Z 551.988,A -85,B 0,C 180,E1 -17264.057,E2 -17264.057} C_VEL
LIN {X 0,Y 307.332,Z 537.48,A -85,B 0,C 180,E1 -17264.906,E2 -17264.906} C_VEL
LIN {X 0,Y 308.674,Z 523.242,A -85,B 0,C 180,E1 -17265.495,E2 -17265.495} C_VEL
LIN {X 0,Y 314.635,Z 422.045,A -85,B 0,C 180,E1 -17268.139,E2 -17268.139} C_VEL
LIN {X 0,Y 308.941,Z 411.263,A -85,B 0,C 180,E1 -17269.643,E2 -17269.643} C_VEL
LIN {X 0,Y 302.685,Z 400.688,A -85,B 0,C 180,E1 -17271.407,E2 -17271.407} C_VEL
LIN {X 0,Y 295.27,Z 389.435,A -85,B 0,C 180,E1 -17273.705,E2 -17273.705} C_VEL
LIN {X 0,Y 291.843,Z 384.704,A -85,B 0,C 180,E1 -17274.862,E2 -17274.862} C_VEL
LIN {X 0,Y 289.152,Z 381.103,A -85,B 0,C 180,E1 -17275.818,E2 -17275.818} C_VEL
LIN {X 0,Y 286.602,Z 378.05,A -85,B 0,C 180,E1 -17276.757,E2 -17276.757} C_VEL
LIN {X 0,Y 285.365,Z 376.069,A -85,B 0,C 180,E1 -17277.264,E2 -17277.264} C_VEL
LIN {X 0,Y 282.872,Z 373.155,A -85,B 0,C 180,E1 -17278.264,E2 -17278.264} C_VEL
LIN {X 0,Y 281.814,Z 371.047,A -85,B 0,C 180,E1 -17278.767,E2 -17278.767} C_VEL
LIN {X 0,Y 279.314,Z 369.019,A -85,B 0,C 180,E1 -17279.819,E2 -17279.819} C_VEL
LIN {X 0,Y 278.016,Z 366.51,A -85,B 0,C 180,E1 -17280.497,E2 -17280.497} C_VEL
LIN {X 0,Y 277.826,Z 365.505,A -85,B 0,C 180,E1 -17280.679,E2 -17280.679} C_VEL
LIN {X 0,Y 277.695,Z 365.518,A -85,B 0,C 180,E1 -17282.901,E2 -17282.901} C_VEL
LIN {X 0,Y 277.604,Z 365.524,A -85,B 0,C 180,E1 -17287.272,E2 -17287.272} C_VEL
LIN {X 0,Y 277.46,Z 365.541,A -85,B 0,C 180,E1 -17290.213,E2 -17290.213} C_VEL
LIN {X 0,Y 277.412,Z 365.553,A -85,B 0,C 180,E1 -17294.675,E2 -17294.675} C_VEL
LIN {X 0,Y 277.337,Z 365.557,A -85,B 0,C 180,E1 -17299.234,E2 -17299.234} C_VEL
LIN {X 0,Y 277.322,Z 365.559,A -85,B 0,C 180,E1 -17304.17,E2 -17304.17} C_VEL
LIN {X 0,Y 277.328,Z 365.559,A -85,B 0,C 180,E1 -17307.505,E2 -17307.505} C_VEL
LIN {X 0,Y 277.274,Z 365.568,A -85,B 0,C 180,E1 -17310.481,E2 -17310.481} C_VEL
LIN {X 0,Y 277.257,Z 365.693,A -85,B 0,C 180,E1 -17313.794,E2 -17313.794} C_VEL
LIN {X 0,Y 278.657,Z 369.015,A -85,B 0,C 180,E1 -17316.188,E2 -17316.188} C_VEL
LIN {X 0,Y 280.761,Z 374.865,A -85,B 0,C 180,E1 -17319.665,E2 -17319.665} C_VEL
LIN {X 0,Y 281.521,Z 376.9,A -85,B 0,C 180,E1 -17320.643,E2 -17320.643} C_VEL
LIN {X 0,Y 286.503,Z 384.202,A -85,B 0,C 180,E1 -17322.711,E2 -17322.711} C_VEL
LIN {X 0,Y 290.682,Z 390.702,A -85,B 0,C 180,E1 -17324.277,E2 -17324.277} C_VEL
LIN {X 0,Y 294.824,Z 397.538,A -85,B 0,C 180,E1 -17325.724,E2 -17325.724} C_VEL
LIN {X 0,Y 298.402,Z 403.753,A -85,B 0,C 180,E1 -17326.896,E2 -17326.896} C_VEL
LIN {X 0,Y 303.534,Z 413.5,A -85,B 0,C 180,E1 -17328.481,E2 -17328.481} C_VEL
LIN {X 0,Y 308.52,Z 424.183,A -85,B 0,C 180,E1 -17329.95,E2 -17329.95} C_VEL
LIN {X 0,Y 311.731,Z 431.842,A -85,B 0,C 180,E1 -17330.856,E2 -17330.856} C_VEL
LIN {X 0,Y 313.463,Z 447.583,A -85,B 0,C 180,E1 -17331.756,E2 -17331.756} C_VEL
LIN {X 0,Y 307.655,Z 548.186,A -85,B 0,C 180,E1 -17334.372,E2 -17334.372} C_VEL
LIN {X 0,Y 305.873,Z 564.065,A -85,B 0,C 180,E1 -17334.991,E2 -17334.991} C_VEL
LIN {X 0,Y 303.534,Z 579.326,A -85,B 0,C 180,E1 -17335.841,E2 -17335.841} C_VEL
LIN {X 0,Y 300.816,Z 593.641,A -85,B 0,C 180,E1 -17336.899,E2 -17336.899} C_VEL
LIN {X 0,Y 297.655,Z 607.842,A -85,B 0,C 180,E1 -17338.247,E2 -17338.247} C_VEL
LIN {X 0,Y 294.222,Z 621.561,A -85,B 0,C 180,E1 -17339.892,E2 -17339.892} C_VEL
LIN {X 0,Y 290.881,Z 633.825,A -85,B 0,C 180,E1 -17341.695,E2 -17341.695} C_VEL
LIN {X 0,Y 287.354,Z 645.925,A -85,B 0,C 180,E1 -17343.88,E2 -17343.88} C_VEL
LIN {X 0,Y 284.499,Z 655.835,A -85,B 0,C 180,E1 -17346.065,E2 -17346.065} C_VEL
LIN {X 0,Y 281.56,Z 665.901,A -85,B 0,C 180,E1 -17348.78,E2 -17348.78} C_VEL
LIN {X 0,Y 279.067,Z 674.51,A -85,B 0,C 180,E1 -17351.651,E2 -17351.651} C_VEL
LIN {X 0,Y 277.317,Z 681.468,A -85,B 0,C 180,E1 -17354.553,E2 -17354.553} C_VEL
LIN {X 0,Y 276.194,Z 687.035,A -85,B 0,C 180,E1 -17357.508,E2 -17357.508} C_VEL
LIN {X 0,Y 275.656,Z 690.265,A -85,B 0,C 180,E1 -17359.719,E2 -17359.719} C_VEL
LIN {X 0,Y 275.367,Z 693.526,A -85,B 0,C 180,E1 -17362.668,E2 -17362.668} C_VEL
LIN {X 0,Y 275.372,Z 695.585,A -85,B 0,C 180,E1 -17365.608,E2 -17365.608} C_VEL
LIN {X 0,Y 275.464,Z 696.411,A -85,B 0,C 180,E1 -17368.537,E2 -17368.537} C_VEL
LIN {X 0,Y 275.578,Z 696.365,A -85,B 0,C 180,E1 -17369.999,E2 -17369.999} C_VEL
LIN {X 0,Y 275.446,Z 695.344,A -85,B 0,C 180,E1 -17372.924,E2 -17372.924} C_VEL
LIN {X 0,Y 275.413,Z 693.093,A -85,B 0,C 180,E1 -17375.858,E2 -17375.858} C_VEL
LIN {X 0,Y 275.527,Z 689.556,A -85,B 0,C 180,E1 -17378.803,E2 -17378.803} C_VEL
LIN {X 0,Y 275.926,Z 684.642,A -85,B 0,C 180,E1 -17381.756,E2 -17381.756} C_VEL
LIN {X 0,Y 276.858,Z 678.231,A -85,B 0,C 180,E1 -17384.705,E2 -17384.705} C_VEL
LIN {X 0,Y 278.349,Z 670.143,A -85,B 0,C 180,E1 -17387.636,E2 -17387.636} C_VEL
LIN {X 0,Y 280.172,Z 661.503,A -85,B 0,C 180,E1 -17390.176,E2 -17390.176} C_VEL
LIN {X 0,Y 282.322,Z 651.714,A -85,B 0,C 180,E1 -17392.546,E2 -17392.546} C_VEL
LIN {X 0,Y 284.748,Z 640.373,A -85,B 0,C 180,E1 -17394.808,E2 -17394.808} C_VEL
LIN {X 0,Y 287.044,Z 629.92,A -85,B 0,C 180,E1 -17396.54,E2 -17396.54} C_VEL
LIN {X 0,Y 289.31,Z 618.804,A -85,B 0,C 180,E1 -17398.077,E2 -17398.077} C_VEL
LIN {X 0,Y 291.552,Z 607.189,A -85,B 0,C 180,E1 -17399.415,E2 -17399.415} C_VEL
LIN {X 0,Y 293.888,Z 593.314,A -85,B 0,C 180,E1 -17400.72,E2 -17400.72} C_VEL
LIN {X 0,Y 295.986,Z 578.68,A -85,B 0,C 180,E1 -17401.791,E2 -17401.791} C_VEL
LIN {X 0,Y 297.807,Z 563.199,A -85,B 0,C 180,E1 -17402.621,E2 -17402.621} C_VEL
LIN {X 0,Y 298.993,Z 548.21,A -85,B 0,C 180,E1 -17403.177,E2 -17403.177} C_VEL
LIN {X 0,Y 303.487,Z 445.966,A -85,B 0,C 180,E1 -17405.777,E2 -17405.777} C_VEL
LIN {X 0,Y 299.818,Z 421.697,A -85,B 0,C 180,E1 -17406.952,E2 -17406.952} C_VEL
LIN {X 0,Y 292.045,Z 403.806,A -85,B 0,C 180,E1 -17408.478,E2 -17408.478} C_VEL
LIN {X 0,Y 284.171,Z 387.162,A -85,B 0,C 180,E1 -17410.081,E2 -17410.081} C_VEL
LIN {X 0,Y 282.248,Z 383.056,A -85,B 0,C 180,E1 -17410.532,E2 -17410.532} C_VEL
LIN {X 0,Y 278.955,Z 371.467,A -85,B 0,C 180,E1 -17414.109,E2 -17414.109} C_VEL
LIN {X 0,Y 277.231,Z 365.58,A -85,B 0,C 180,E1 -17416.083,E2 -17416.083} C_VEL
LIN {X 0,Y 277.231,Z 365.576,A -85,B 0,C 180,E1 -17420.672,E2 -17420.672} C_VEL
LIN {X 0,Y 277.281,Z 365.574,A -85,B 0,C 180,E1 -17424.341,E2 -17424.341} C_VEL
LIN {X 0,Y 277.241,Z 365.575,A -85,B 0,C 180,E1 -17427.836,E2 -17427.836} C_VEL
LIN {X 0,Y 277.286,Z 365.571,A -85,B 0,C 180,E1 -17431.213,E2 -17431.213} C_VEL
LIN {X 0,Y 277.31,Z 365.563,A -85,B 0,C 180,E1 -17434.48,E2 -17434.48} C_VEL
LIN {X 0,Y 277.282,Z 365.567,A -85,B 0,C 180,E1 -17437.655,E2 -17437.655} C_VEL
LIN {X 0,Y 277.342,Z 365.565,A -85,B 0,C 180,E1 -17440.766,E2 -17440.766} C_VEL
LIN {X 0,Y 277.432,Z 365.55,A -85,B 0,C 180,E1 -17445.326,E2 -17445.326} C_VEL
LIN {X 0,Y 277.504,Z 365.523,A -85,B 0,C 180,E1 -17449.789,E2 -17449.789} C_VEL
LIN {X 0,Y 277.646,Z 365.521,A -85,B 0,C 180,E1 -17452.729,E2 -17452.729} C_VEL
LIN {X 0,Y 277.819,Z 365.491,A -85,B 0,C 180,E1 -17458.551,E2 -17458.551} C_VEL
LIN {X 0,Y 277.819,Z 365.502,A -85,B 0,C 180,E1 -17461.45,E2 -17461.45} C_VEL
LIN {X 0,Y 277.651,Z 365.511,A -85,B 0,C 180,E1 -17467.272,E2 -17467.272} C_VEL
LIN {X 0,Y 277.505,Z 365.539,A -85,B 0,C 180,E1 -17470.212,E2 -17470.212} C_VEL
LIN {X 0,Y 277.433,Z 365.544,A -85,B 0,C 180,E1 -17474.675,E2 -17474.675} C_VEL
LIN {X 0,Y 277.343,Z 365.561,A -85,B 0,C 180,E1 -17479.235,E2 -17479.235} C_VEL
LIN {X 0,Y 277.29,Z 365.563,A -85,B 0,C 180,E1 -17484.158,E2 -17484.158} C_VEL
LIN {X 0,Y 277.323,Z 365.558,A -85,B 0,C 180,E1 -17487.505,E2 -17487.505} C_VEL
LIN {X 0,Y 277.271,Z 365.573,A -85,B 0,C 180,E1 -17490.482,E2 -17490.482} C_VEL
LIN {X 0,Y 277.246,Z 365.565,A -85,B 0,C 180,E1 -17493.897,E2 -17493.897} C_VEL
LIN {X 0,Y 277.267,Z 365.568,A -85,B 0,C 180,E1 -17497.47,E2 -17497.47} C_VEL
LIN {X 0,Y 277.209,Z 365.574,A -85,B 0,C 180,E1 -17501.237,E2 -17501.237} C_VEL
LIN {X 0,Y 277.2,Z 365.576,A -85,B 0,C 180,E1 -17505.228,E2 -17505.228} C_VEL
LIN {X 0,Y 277.222,Z 365.573,A -85,B 0,C 180,E1 -17509.513,E2 -17509.513} C_VEL
LIN {X 0,Y 277.265,Z 365.566,A -85,B 0,C 180,E1 -17512.531,E2 -17512.531} C_VEL
LIN {X 0,Y 277.247,Z 365.575,A -85,B 0,C 180,E1 -17516.105,E2 -17516.105} C_VEL
LIN {X 0,Y 277.263,Z 365.568,A -85,B 0,C 180,E1 -17519.54,E2 -17519.54} C_VEL
LIN {X 0,Y 277.298,Z 365.564,A -85,B 0,C 180,E1 -17522.858,E2 -17522.858} C_VEL
LIN {X 0,Y 277.289,Z 365.567,A -85,B 0,C 180,E1 -17526.077,E2 -17526.077} C_VEL
LIN {X 0,Y 277.302,Z 365.568,A -85,B 0,C 180,E1 -17530.764,E2 -17530.764} C_VEL
LIN {X 0,Y 277.374,Z 365.557,A -85,B 0,C 180,E1 -17535.323,E2 -17535.323} C_VEL
LIN {X 0,Y 277.458,Z 365.548,A -85,B 0,C 180,E1 -17539.788,E2 -17539.788} C_VEL
LIN {X 0,Y 277.604,Z 365.532,A -85,B 0,C 180,E1 -17542.728,E2 -17542.728} C_VEL
LIN {X 0,Y 277.808,Z 365.506,A -85,B 0,C 180,E1 -17548.551,E2 -17548.551} C_VEL
LIN {X 0,Y 277.816,Z 365.717,A -85,B 0,C 180,E1 -17549.321,E2 -17549.321} C_VEL
LIN {X 0,Y 278.736,Z 368.264,A -85,B 0,C 180,E1 -17549.547,E2 -17549.547} C_VEL
LIN {X 0,Y 280.441,Z 370.97,A -85,B 0,C 180,E1 -17549.888,E2 -17549.888} C_VEL
LIN {X 0,Y 286.266,Z 381.237,A -85,B 0,C 180,E1 -17551.055,E2 -17551.055} C_VEL
LIN {X 0,Y 296.956,Z 400.755,A -85,B 0,C 180,E1 -17553.087,E2 -17553.087} C_VEL
LIN {X 0,Y 304.111,Z 415.471,A -85,B 0,C 180,E1 -17554.392,E2 -17554.392} C_VEL
LIN {X 0,Y 299.539,Z 519.572,A -85,B 0,C 180,E1 -17557.048,E2 -17557.048} C_VEL
LIN {X 0,Y 298.347,Z 535.704,A -85,B 0,C 180,E1 -17557.726,E2 -17557.726} C_VEL
LIN {X 0,Y 296.712,Z 551.463,A -85,B 0,C 180,E1 -17558.685,E2 -17558.685} C_VEL
LIN {X 0,Y 294.918,Z 565.035,A -85,B 0,C 180,E1 -17559.765,E2 -17559.765} C_VEL
LIN {X 0,Y 292.591,Z 579.734,A -85,B 0,C 180,E1 -17561.255,E2 -17561.255} C_VEL
LIN {X 0,Y 290.2,Z 592.714,A -85,B 0,C 180,E1 -17562.885,E2 -17562.885} C_VEL
LIN {X 0,Y 287.815,Z 604.449,A -85,B 0,C 180,E1 -17564.676,E2 -17564.676} C_VEL
LIN {X 0,Y 285.437,Z 615.664,A -85,B 0,C 180,E1 -17566.75,E2 -17566.75} C_VEL
LIN {X 0,Y 283.288,Z 624.988,A -85,B 0,C 180,E1 -17568.816,E2 -17568.816} C_VEL
LIN {X 0,Y 281.193,Z 634.137,A -85,B 0,C 180,E1 -17571.249,E2 -17571.249} C_VEL
LIN {X 0,Y 279.463,Z 641.82,A -85,B 0,C 180,E1 -17573.727,E2 -17573.727} C_VEL
LIN {X 0,Y 278.052,Z 648.267,A -85,B 0,C 180,E1 -17576.253,E2 -17576.253} C_VEL
LIN {X 0,Y 277.017,Z 653.59,A -85,B 0,C 180,E1 -17578.819,E2 -17578.819} C_VEL
LIN {X 0,Y 276.28,Z 657.833,A -85,B 0,C 180,E1 -17581.432,E2 -17581.432} C_VEL
LIN {X 0,Y 275.664,Z 661.094,A -85,B 0,C 180,E1 -17584.118,E2 -17584.118} C_VEL
LIN {X 0,Y 275.372,Z 662.74,A -85,B 0,C 180,E1 -17585.945,E2 -17585.945} C_VEL
LIN {X 0,Y 275.223,Z 663.941,A -85,B 0,C 180,E1 -17587.797,E2 -17587.797} C_VEL
LIN {X 0,Y 275.203,Z 664.737,A -85,B 0,C 180,E1 -17589.992,E2 -17589.992} C_VEL
LIN {X 0,Y 275.298,Z 664.878,A -85,B 0,C 180,E1 -17592.239,E2 -17592.239} C_VEL
LIN {X 0,Y 275.522,Z 664.42,A -85,B 0,C 180,E1 -17594.419,E2 -17594.419} C_VEL
LIN {X 0,Y 276.206,Z 662.583,A -85,B 0,C 180,E1 -17597.554,E2 -17597.554} C_VEL
LIN {X 0,Y 277.24,Z 659.403,A -85,B 0,C 180,E1 -17600.672,E2 -17600.672} C_VEL
LIN {X 0,Y 278.691,Z 654.769,A -85,B 0,C 180,E1 -17603.802,E2 -17603.802} C_VEL
LIN {X 0,Y 280.481,Z 649.337,A -85,B 0,C 180,E1 -17606.546,E2 -17606.546} C_VEL
LIN {X 0,Y 282.797,Z 642.276,A -85,B 0,C 180,E1 -17609.372,E2 -17609.372} C_VEL
LIN {X 0,Y 285.667,Z 633.596,A -85,B 0,C 180,E1 -17612.131,E2 -17612.131} C_VEL
LIN {X 0,Y 288.49,Z 625.005,A -85,B 0,C 180,E1 -17614.34,E2 -17614.34} C_VEL
LIN {X 0,Y 291.621,Z 614.516,A -85,B 0,C 180,E1 -17616.583,E2 -17616.583} C_VEL
LIN {X 0,Y 294.929,Z 602.707,A -85,B 0,C 180,E1 -17618.643,E2 -17618.643} C_VEL
LIN {X 0,Y 297.893,Z 591.317,A -85,B 0,C 180,E1 -17620.273,E2 -17620.273} C_VEL
LIN {X 0,Y 300.886,Z 578.342,A -85,B 0,C 180,E1 -17621.795,E2 -17621.795} C_VEL
LIN {X 0,Y 303.262,Z 565.985,A -85,B 0,C 180,E1 -17622.987,E2 -17622.987} C_VEL
LIN {X 0,Y 303.628,Z 560.735,A -85,B 0,C 180,E1 -17623.512,E2 -17623.512} C_VEL
LIN {X 0,Y 301.821,Z 545.526,A -85,B 0,C 180,E1 -17625.259,E2 -17625.259} C_VEL
LIN {X 0,Y 301.798,Z 540.077,A -85,B 0,C 180,E1 -17625.677,E2 -17625.677} C_VEL
LIN {X 0,Y 301.992,Z 538.193,A -85,B 0,C 180,E1 -17625.772,E2 -17625.772} C_VEL
LIN {X 0,Y 303.469,Z 523.002,A -85,B 0,C 180,E1 -17626.408,E2 -17626.408} C_VEL
LIN {X 0,Y 309.454,Z 424.631,A -85,B 0,C 180,E1 -17629.021,E2 -17629.021} C_VEL
LIN {X 0,Y 302.969,Z 412.408,A -85,B 0,C 180,E1 -17630.856,E2 -17630.856} C_VEL
LIN {X 0,Y 296.932,Z 402.514,A -85,B 0,C 180,E1 -17632.686,E2 -17632.686} C_VEL
LIN {X 0,Y 291.425,Z 394.182,A -85,B 0,C 180,E1 -17634.507,E2 -17634.507} C_VEL
LIN {X 0,Y 288.774,Z 390.419,A -85,B 0,C 180,E1 -17635.45,E2 -17635.45} C_VEL
LIN {X 0,Y 286.338,Z 387.14,A -85,B 0,C 180,E1 -17636.343,E2 -17636.343} C_VEL
LIN {X 0,Y 283.531,Z 383.482,A -85,B 0,C 180,E1 -17637.447,E2 -17637.447} C_VEL
LIN {X 0,Y 282.488,Z 381.975,A -85,B 0,C 180,E1 -17637.883,E2 -17637.883} C_VEL
LIN {X 0,Y 279.975,Z 378.606,A -85,B 0,C 180,E1 -17638.971,E2 -17638.971} C_VEL
LIN {X 0,Y 279.12,Z 377.303,A -85,B 0,C 180,E1 -17639.368,E2 -17639.368} C_VEL
LIN {X 0,Y 276.729,Z 374.899,A -85,B 0,C 180,E1 -17640.454,E2 -17640.454} C_VEL
LIN {X 0,Y 275.216,Z 372.083,A -85,B 0,C 180,E1 -17641.28,E2 -17641.28} C_VEL
LIN {X 0,Y 272.555,Z 370.4,A -85,B 0,C 180,E1 -17642.6,E2 -17642.6} C_VEL
LIN {X 0,Y 270.895,Z 367.963,A -85,B 0,C 180,E1 -17643.625,E2 -17643.625} C_VEL
LIN {X 0,Y 270.449,Z 366.417,A -85,B 0,C 180,E1 -17644.004,E2 -17644.004} C_VEL
LIN {X 0,Y 270.566,Z 366.401,A -85,B 0,C 180,E1 -17647.462,E2 -17647.462} C_VEL
LIN {X 0,Y 270.413,Z 366.42,A -85,B 0,C 180,E1 -17650.482,E2 -17650.482} C_VEL
LIN {X 0,Y 270.38,Z 366.424,A -85,B 0,C 180,E1 -17655.065,E2 -17655.065} C_VEL
LIN {X 0,Y 270.299,Z 366.437,A -85,B 0,C 180,E1 -17659.755,E2 -17659.755} C_VEL
LIN {X 0,Y 270.277,Z 366.436,A -85,B 0,C 180,E1 -17664.585,E2 -17664.585} C_VEL
LIN {X 0,Y 270.274,Z 366.44,A -85,B 0,C 180,E1 -17667.908,E2 -17667.908} C_VEL
LIN {X 0,Y 270.237,Z 366.588,A -85,B 0,C 180,E1 -17670.731,E2 -17670.731} C_VEL
LIN {X 0,Y 272.505,Z 372.441,A -85,B 0,C 180,E1 -17675.47,E2 -17675.47} C_VEL
LIN {X 0,Y 273.805,Z 375.696,A -85,B 0,C 180,E1 -17677.524,E2 -17677.524} C_VEL
LIN {X 0,Y 279.245,Z 383.435,A -85,B 0,C 180,E1 -17680.219,E2 -17680.219} C_VEL
LIN {X 0,Y 283.754,Z 390.247,A -85,B 0,C 180,E1 -17682.167,E2 -17682.167} C_VEL
LIN {X 0,Y 287.564,Z 396.298,A -85,B 0,C 180,E1 -17683.663,E2 -17683.663} C_VEL
LIN {X 0,Y 291.875,Z 403.626,A -85,B 0,C 180,E1 -17685.242,E2 -17685.242} C_VEL
LIN {X 0,Y 296.603,Z 412.143,A -85,B 0,C 180,E1 -17686.834,E2 -17686.834} C_VEL
LIN {X 0,Y 302.421,Z 424.146,A -85,B 0,C 180,E1 -17688.678,E2 -17688.678} C_VEL
LIN {X 0,Y 306.892,Z 434.922,A -85,B 0,C 180,E1 -17690.043,E2 -17690.043} C_VEL
LIN {X 0,Y 308.389,Z 448.745,A -85,B 0,C 180,E1 -17690.86,E2 -17690.86} C_VEL
LIN {X 0,Y 302.331,Z 548.14,A -85,B 0,C 180,E1 -17693.49,E2 -17693.49} C_VEL
LIN {X 0,Y 300.494,Z 563.783,A -85,B 0,C 180,E1 -17694.114,E2 -17694.114} C_VEL
LIN {X 0,Y 297.947,Z 579.531,A -85,B 0,C 180,E1 -17695.006,E2 -17695.006} C_VEL
LIN {X 0,Y 295.322,Z 592.831,A -85,B 0,C 180,E1 -17695.996,E2 -17695.996} C_VEL
LIN {X 0,Y 292.188,Z 606.575,A -85,B 0,C 180,E1 -17697.304,E2 -17697.304} C_VEL
LIN {X 0,Y 288.793,Z 619.656,A -85,B 0,C 180,E1 -17698.859,E2 -17698.859} C_VEL
LIN {X 0,Y 285.237,Z 632.092,A -85,B 0,C 180,E1 -17700.678,E2 -17700.678} C_VEL
LIN {X 0,Y 281.5,Z 644.391,A -85,B 0,C 180,E1 -17702.894,E2 -17702.894} C_VEL
LIN {X 0,Y 278.388,Z 654.456,A -85,B 0,C 180,E1 -17705.116,E2 -17705.116} C_VEL
LIN {X 0,Y 275.633,Z 663.437,A -85,B 0,C 180,E1 -17707.513,E2 -17707.513} C_VEL
LIN {X 0,Y 273.145,Z 671.381,A -85,B 0,C 180,E1 -17710.066,E2 -17710.066} C_VEL
LIN {X 0,Y 271.251,Z 678.026,A -85,B 0,C 180,E1 -17712.664,E2 -17712.664} C_VEL
LIN {X 0,Y 269.711,Z 684.201,A -85,B 0,C 180,E1 -17715.667,E2 -17715.667} C_VEL
LIN {X 0,Y 268.736,Z 689.019,A -85,B 0,C 180,E1 -17718.688,E2 -17718.688} C_VEL
LIN {X 0,Y 268.395,Z 691.74,A -85,B 0,C 180,E1 -17720.96,E2 -17720.96} C_VEL
LIN {X 0,Y 268.29,Z 694.348,A -85,B 0,C 180,E1 -17723.985,E2 -17723.985} C_VEL
LIN {X 0,Y 268.353,Z 695.764,A -85,B 0,C 180,E1 -17726.997,E2 -17726.997} C_VEL
LIN {X 0,Y 268.489,Z 695.94,A -85,B 0,C 180,E1 -17729.999,E2 -17729.999} C_VEL
LIN {X 0,Y 268.372,Z 694.874,A -85,B 0,C 180,E1 -17733.002,E2 -17733.002} C_VEL
LIN {X 0,Y 268.333,Z 692.573,A -85,B 0,C 180,E1 -17736.013,E2 -17736.013} C_VEL
LIN {X 0,Y 268.441,Z 688.981,A -85,B 0,C 180,E1 -17739.037,E2 -17739.037} C_VEL
LIN {X 0,Y 268.922,Z 684.011,A -85,B 0,C 180,E1 -17742.067,E2 -17742.067} C_VEL
LIN {X 0,Y 269.895,Z 677.533,A -85,B 0,C 180,E1 -17745.093,E2 -17745.093} C_VEL
LIN {X 0,Y 271.251,Z 670.523,A -85,B 0,C 180,E1 -17747.724,E2 -17747.724} C_VEL
LIN {X 0,Y 273.089,Z 662.041,A -85,B 0,C 180,E1 -17750.329,E2 -17750.329} C_VEL
LIN {X 0,Y 275.343,Z 652.315,A -85,B 0,C 180,E1 -17752.781,E2 -17752.781} C_VEL
LIN {X 0,Y 277.775,Z 641.294,A -85,B 0,C 180,E1 -17755.074,E2 -17755.074} C_VEL
LIN {X 0,Y 280.366,Z 629.883,A -85,B 0,C 180,E1 -17757.022,E2 -17757.022} C_VEL
LIN {X 0,Y 282.697,Z 618.827,A -85,B 0,C 180,E1 -17758.591,E2 -17758.591} C_VEL
LIN {X 0,Y 285.25,Z 606.101,A -85,B 0,C 180,E1 -17760.081,E2 -17760.081} C_VEL
LIN {X 0,Y 287.732,Z 591.338,A -85,B 0,C 180,E1 -17761.472,E2 -17761.472} C_VEL
LIN {X 0,Y 289.915,Z 576.52,A -85,B 0,C 180,E1 -17762.537,E2 -17762.537} C_VEL
LIN {X 0,Y 291.672,Z 561.245,A -85,B 0,C 180,E1 -17763.344,E2 -17763.344} C_VEL
LIN {X 0,Y 292.898,Z 545.386,A -85,B 0,C 180,E1 -17763.908,E2 -17763.908} C_VEL
LIN {X 0,Y 297.324,Z 446.462,A -85,B 0,C 180,E1 -17766.472,E2 -17766.472} C_VEL
LIN {X 0,Y 294.141,Z 424.736,A -85,B 0,C 180,E1 -17767.538,E2 -17767.538} C_VEL
LIN {X 0,Y 286.59,Z 407.2,A -85,B 0,C 180,E1 -17769.078,E2 -17769.078} C_VEL
LIN {X 0,Y 278.614,Z 390.389,A -85,B 0,C 180,E1 -17770.753,E2 -17770.753} C_VEL
LIN {X 0,Y 274.895,Z 382.644,A -85,B 0,C 180,E1 -17771.606,E2 -17771.606} C_VEL
LIN {X 0,Y 271.282,Z 370.23,A -85,B 0,C 180,E1 -17775.615,E2 -17775.615} C_VEL
LIN {X 0,Y 270.175,Z 366.453,A -85,B 0,C 180,E1 -17776.974,E2 -17776.974} C_VEL
LIN {X 0,Y 270.203,Z 366.445,A -85,B 0,C 180,E1 -17781.374,E2 -17781.374} C_VEL
LIN {X 0,Y 270.198,Z 366.454,A -85,B 0,C 180,E1 -17785.095,E2 -17785.095} C_VEL
LIN {X 0,Y 270.197,Z 366.458,A -85,B 0,C 180,E1 -17789.131,E2 -17789.131} C_VEL
LIN {X 0,Y 270.261,Z 366.445,A -85,B 0,C 180,E1 -17792.146,E2 -17792.146} C_VEL
LIN {X 0,Y 270.274,Z 366.444,A -85,B 0,C 180,E1 -17795.519,E2 -17795.519} C_VEL
LIN {X 0,Y 270.298,Z 366.44,A -85,B 0,C 180,E1 -17800.245,E2 -17800.245} C_VEL
LIN {X 0,Y 270.4,Z 366.43,A -85,B 0,C 180,E1 -17804.936,E2 -17804.936} C_VEL
LIN {X 0,Y 270.439,Z 366.4,A -85,B 0,C 180,E1 -17809.519,E2 -17809.519} C_VEL
LIN {X 0,Y 270.605,Z 366.396,A -85,B 0,C 180,E1 -17812.539,E2 -17812.539} C_VEL
LIN {X 0,Y 270.785,Z 366.366,A -85,B 0,C 180,E1 -17818.513,E2 -17818.513} C_VEL
LIN {X 0,Y 270.785,Z 366.378,A -85,B 0,C 180,E1 -17821.488,E2 -17821.488} C_VEL
LIN {X 0,Y 270.609,Z 366.387,A -85,B 0,C 180,E1 -17827.462,E2 -17827.462} C_VEL
LIN {X 0,Y 270.44,Z 366.42,A -85,B 0,C 180,E1 -17830.482,E2 -17830.482} C_VEL
LIN {X 0,Y 270.401,Z 366.415,A -85,B 0,C 180,E1 -17835.065,E2 -17835.065} C_VEL
LIN {X 0,Y 270.3,Z 366.437,A -85,B 0,C 180,E1 -17839.756,E2 -17839.756} C_VEL
LIN {X 0,Y 270.236,Z 366.436,A -85,B 0,C 180,E1 -17844.59,E2 -17844.59} C_VEL
LIN {X 0,Y 270.27,Z 366.436,A -85,B 0,C 180,E1 -17847.909,E2 -17847.909} C_VEL
LIN {X 0,Y 270.183,Z 366.452,A -85,B 0,C 180,E1 -17851.349,E2 -17851.349} C_VEL
LIN {X 0,Y 270.201,Z 366.438,A -85,B 0,C 180,E1 -17854.906,E2 -17854.906} C_VEL
LIN {X 0,Y 270.197,Z 366.455,A -85,B 0,C 180,E1 -17858.711,E2 -17858.711} C_VEL
LIN {X 0,Y 270.171,Z 366.445,A -85,B 0,C 180,E1 -17862.559,E2 -17862.559} C_VEL
LIN {X 0,Y 270.165,Z 366.459,A -85,B 0,C 180,E1 -17866.752,E2 -17866.752} C_VEL
LIN {X 0,Y 270.198,Z 366.44,A -85,B 0,C 180,E1 -17871.291,E2 -17871.291} C_VEL
LIN {X 0,Y 270.202,Z 366.452,A -85,B 0,C 180,E1 -17875.096,E2 -17875.096} C_VEL
LIN {X 0,Y 270.185,Z 366.449,A -85,B 0,C 180,E1 -17879.137,E2 -17879.137} C_VEL
LIN {X 0,Y 270.225,Z 366.451,A -85,B 0,C 180,E1 -17882.163,E2 -17882.163} C_VEL
LIN {X 0,Y 270.232,Z 366.444,A -85,B 0,C 180,E1 -17885.542,E2 -17885.542} C_VEL
LIN {X 0,Y 270.252,Z 366.44,A -85,B 0,C 180,E1 -17890.241,E2 -17890.241} C_VEL
LIN {X 0,Y 270.341,Z 366.433,A -85,B 0,C 180,E1 -17894.933,E2 -17894.933} C_VEL
LIN {X 0,Y 270.409,Z 366.425,A -85,B 0,C 180,E1 -17899.518,E2 -17899.518} C_VEL
LIN {X 0,Y 270.566,Z 366.406,A -85,B 0,C 180,E1 -17902.538,E2 -17902.538} C_VEL
LIN {X 0,Y 270.72,Z 366.387,A -85,B 0,C 180,E1 -17908.234,E2 -17908.234} C_VEL
LIN {X 0,Y 271.815,Z 369.276,A -85,B 0,C 180,E1 -17908.543,E2 -17908.543} C_VEL
LIN {X 0,Y 273.319,Z 371.616,A -85,B 0,C 180,E1 -17908.858,E2 -17908.858} C_VEL
LIN {X 0,Y 280.64,Z 384.274,A -85,B 0,C 180,E1 -17910.381,E2 -17910.381} C_VEL
LIN {X 0,Y 292.052,Z 405.323,A -85,B 0,C 180,E1 -17912.617,E2 -17912.617} C_VEL
LIN {X 0,Y 298.037,Z 417.716,A -85,B 0,C 180,E1 -17913.749,E2 -17913.749} C_VEL
LIN {X 0,Y 293.249,Z 520.738,A -85,B 0,C 180,E1 -17916.429,E2 -17916.429} C_VEL
LIN {X 0,Y 292.052,Z 536.161,A -85,B 0,C 180,E1 -17917.095,E2 -17917.095} C_VEL
LIN {X 0,Y 290.503,Z 550.995,A -85,B 0,C 180,E1 -17918.007,E2 -17918.007} C_VEL
LIN {X 0,Y 288.455,Z 565.781,A -85,B 0,C 180,E1 -17919.201,E2 -17919.201} C_VEL
LIN {X 0,Y 286.099,Z 580.254,A -85,B 0,C 180,E1 -17920.701,E2 -17920.701} C_VEL
LIN {X 0,Y 283.652,Z 593.059,A -85,B 0,C 180,E1 -17922.34,E2 -17922.34} C_VEL
LIN {X 0,Y 281.13,Z 605.126,A -85,B 0,C 180,E1 -17924.226,E2 -17924.226} C_VEL
LIN {X 0,Y 278.926,Z 615.074,A -85,B 0,C 180,E1 -17926.092,E2 -17926.092} C_VEL
LIN {X 0,Y 276.793,Z 624.207,A -85,B 0,C 180,E1 -17928.122,E2 -17928.122} C_VEL
LIN {X 0,Y 274.554,Z 633.568,A -85,B 0,C 180,E1 -17930.609,E2 -17930.609} C_VEL
LIN {X 0,Y 272.755,Z 641.408,A -85,B 0,C 180,E1 -17933.138,E2 -17933.138} C_VEL
LIN {X 0,Y 270.986,Z 648.995,A -85,B 0,C 180,E1 -17936.162,E2 -17936.162} C_VEL
LIN {X 0,Y 269.935,Z 654.249,A -85,B 0,C 180,E1 -17938.795,E2 -17938.795} C_VEL
LIN {X 0,Y 269.165,Z 658.469,A -85,B 0,C 180,E1 -17941.481,E2 -17941.481} C_VEL
LIN {X 0,Y 268.741,Z 660.727,A -85,B 0,C 180,E1 -17943.312,E2 -17943.312} C_VEL
LIN {X 0,Y 268.314,Z 662.954,A -85,B 0,C 180,E1 -17945.708,E2 -17945.708} C_VEL
LIN {X 0,Y 268.093,Z 664.819,A -85,B 0,C 180,E1 -17948.989,E2 -17948.989} C_VEL
LIN {X 0,Y 268.146,Z 665.282,A -85,B 0,C 180,E1 -17950.939,E2 -17950.939} C_VEL
LIN {X 0,Y 268.281,Z 665.272,A -85,B 0,C 180,E1 -17952.931,E2 -17952.931} C_VEL
LIN {X 0,Y 268.541,Z 664.685,A -85,B 0,C 180,E1 -17955.039,E2 -17955.039} C_VEL
LIN {X 0,Y 269.034,Z 663.466,A -85,B 0,C 180,E1 -17957.218,E2 -17957.218} C_VEL
LIN {X 0,Y 270.048,Z 660.641,A -85,B 0,C 180,E1 -17960.359,E2 -17960.359} C_VEL
LIN {X 0,Y 271.431,Z 656.534,A -85,B 0,C 180,E1 -17963.449,E2 -17963.449} C_VEL
LIN {X 0,Y 273.331,Z 651.06,A -85,B 0,C 180,E1 -17966.493,E2 -17966.493} C_VEL
LIN {X 0,Y 275.642,Z 644.461,A -85,B 0,C 180,E1 -17969.34,E2 -17969.34} C_VEL
LIN {X 0,Y 278.462,Z 636.541,A -85,B 0,C 180,E1 -17972.051,E2 -17972.051} C_VEL
LIN {X 0,Y 281.605,Z 627.459,A -85,B 0,C 180,E1 -17974.562,E2 -17974.562} C_VEL
LIN {X 0,Y 284.976,Z 616.92,A -85,B 0,C 180,E1 -17976.951,E2 -17976.951} C_VEL
LIN {X 0,Y 288.136,Z 606.397,A -85,B 0,C 180,E1 -17978.913,E2 -17978.913} C_VEL
LIN {X 0,Y 291.67,Z 593.726,A -85,B 0,C 180,E1 -17980.828,E2 -17980.828} C_VEL
LIN {X 0,Y 294.863,Z 580.597,A -85,B 0,C 180,E1 -17982.44,E2 -17982.44} C_VEL
LIN {X 0,Y 297.677,Z 566.864,A -85,B 0,C 180,E1 -17983.798,E2 -17983.798} C_VEL
LIN {X 0,Y 300.041,Z 552.997,A -85,B 0,C 180,E1 -17984.885,E2 -17984.885} C_VEL
LIN {X 0,Y 301.992,Z 538.193,A -85,B 0,C 180,E1 -17985.772,E2 -17985.772} C_VEL
LIN {X 0,Y 302.272,Z 532.548,A -85,B 0,C 180,E1 -17986.096,E2 -17986.096} C_VEL
LIN {X 0,Y 301.054,Z 523.489,A -85,B 0,C 180,E1 -17986.822,E2 -17986.822} C_VEL
LIN {X 0,Y 299.451,Z 514.37,A -85,B 0,C 180,E1 -17987.505,E2 -17987.505} C_VEL
LIN {X 0,Y 299.246,Z 508.623,A -85,B 0,C 180,E1 -17987.76,E2 -17987.76} C_VEL
LIN {X 0,Y 304.483,Z 427.461,A -85,B 0,C 180,E1 -17989.919,E2 -17989.919} C_VEL
LIN {X 0,Y 297.48,Z 414.41,A -85,B 0,C 180,E1 -17992.022,E2 -17992.022} C_VEL
LIN {X 0,Y 291.16,Z 404.157,A -85,B 0,C 180,E1 -17994.089,E2 -17994.089} C_VEL
LIN {X 0,Y 286.224,Z 396.727,A -85,B 0,C 180,E1 -17995.872,E2 -17995.872} C_VEL
LIN {X 0,Y 283.223,Z 392.707,A -85,B 0,C 180,E1 -17997.028,E2 -17997.028} C_VEL
LIN {X 0,Y 280.562,Z 388.962,A -85,B 0,C 180,E1 -17998.134,E2 -17998.134} C_VEL
LIN {X 0,Y 277.231,Z 384.323,A -85,B 0,C 180,E1 -17999.636,E2 -17999.636} C_VEL
LIN {X 0,Y 274.031,Z 380.499,A -85,B 0,C 180,E1 -18001.193,E2 -18001.193} C_VEL
LIN {X 0,Y 273.042,Z 378.704,A -85,B 0,C 180,E1 -18001.748,E2 -18001.748} C_VEL
LIN {X 0,Y 270.229,Z 376.477,A -85,B 0,C 180,E1 -18003.261,E2 -18003.261} C_VEL
LIN {X 0,Y 268.564,Z 373.704,A -85,B 0,C 180,E1 -18004.361,E2 -18004.361} C_VEL
LIN {X 0,Y 268.378,Z 373.197,A -85,B 0,C 180,E1 -18004.505,E2 -18004.505} C_VEL
LIN {X 0,Y 265.86,Z 371.751,A -85,B 0,C 180,E1 -18006.069,E2 -18006.069} C_VEL
LIN {X 0,Y 264.122,Z 369.39,A -85,B 0,C 180,E1 -18007.501,E2 -18007.501} C_VEL
LIN {X 0,Y 263.493,Z 367.286,A -85,B 0,C 180,E1 -18008.242,E2 -18008.242} C_VEL
LIN {X 0,Y 263.321,Z 367.303,A -85,B 0,C 180,E1 -18012.328,E2 -18012.328} C_VEL
LIN {X 0,Y 263.303,Z 367.303,A -85,B 0,C 180,E1 -18016.073,E2 -18016.073} C_VEL
LIN {X 0,Y 263.264,Z 367.317,A -85,B 0,C 180,E1 -18020.306,E2 -18020.306} C_VEL
LIN {X 0,Y 263.211,Z 367.32,A -85,B 0,C 180,E1 -18025.29,E2 -18025.29} C_VEL
LIN {X 0,Y 263.234,Z 367.534,A -85,B 0,C 180,E1 -18026.564,E2 -18026.564} C_VEL
LIN {X 0,Y 264.542,Z 370.69,A -85,B 0,C 180,E1 -18030.315,E2 -18030.315} C_VEL
LIN {X 0,Y 265.869,Z 374.151,A -85,B 0,C 180,E1 -18033.321,E2 -18033.321} C_VEL
LIN {X 0,Y 271.838,Z 382.408,A -85,B 0,C 180,E1 -18037.141,E2 -18037.141} C_VEL
LIN {X 0,Y 276.9,Z 389.817,A -85,B 0,C 180,E1 -18039.745,E2 -18039.745} C_VEL
LIN {X 0,Y 280.913,Z 396.017,A -85,B 0,C 180,E1 -18041.557,E2 -18041.557} C_VEL
LIN {X 0,Y 284.688,Z 402.283,A -85,B 0,C 180,E1 -18043.122,E2 -18043.122} C_VEL
LIN {X 0,Y 288.297,Z 408.514,A -85,B 0,C 180,E1 -18044.495,E2 -18044.495} C_VEL
LIN {X 0,Y 292.621,Z 416.464,A -85,B 0,C 180,E1 -18046.043,E2 -18046.043} C_VEL
LIN {X 0,Y 298.686,Z 429.362,A -85,B 0,C 180,E1 -18048.076,E2 -18048.076} C_VEL
LIN {X 0,Y 302.314,Z 438.624,A -85,B 0,C 180,E1 -18049.246,E2 -18049.246} C_VEL
LIN {X 0,Y 303.405,Z 450.166,A -85,B 0,C 180,E1 -18049.937,E2 -18049.937} C_VEL
LIN {X 0,Y 297.194,Z 547.408,A -85,B 0,C 180,E1 -18052.54,E2 -18052.54} C_VEL
LIN {X 0,Y 295.304,Z 563.117,A -85,B 0,C 180,E1 -18053.169,E2 -18053.169} C_VEL
LIN {X 0,Y 292.936,Z 577.736,A -85,B 0,C 180,E1 -18053.999,E2 -18053.999} C_VEL
LIN {X 0,Y 289.914,Z 592.13,A -85,B 0,C 180,E1 -18055.06,E2 -18055.06} C_VEL
LIN {X 0,Y 286.683,Z 605.778,A -85,B 0,C 180,E1 -18056.376,E2 -18056.376} C_VEL
LIN {X 0,Y 282.773,Z 620.191,A -85,B 0,C 180,E1 -18058.119,E2 -18058.119} C_VEL
LIN {X 0,Y 279.08,Z 632.488,A -85,B 0,C 180,E1 -18059.966,E2 -18059.966} C_VEL
LIN {X 0,Y 275.172,Z 644.624,A -85,B 0,C 180,E1 -18062.217,E2 -18062.217} C_VEL
LIN {X 0,Y 272.021,Z 654.237,A -85,B 0,C 180,E1 -18064.398,E2 -18064.398} C_VEL
LIN {X 0,Y 269.039,Z 663.441,A -85,B 0,C 180,E1 -18066.93,E2 -18066.93} C_VEL
LIN {X 0,Y 266.098,Z 672.354,A -85,B 0,C 180,E1 -18069.918,E2 -18069.918} C_VEL
LIN {X 0,Y 263.936,Z 679.567,A -85,B 0,C 180,E1 -18072.967,E2 -18072.967} C_VEL
LIN {X 0,Y 262.431,Z 685.299,A -85,B 0,C 180,E1 -18076.052,E2 -18076.052} C_VEL
LIN {X 0,Y 261.547,Z 689.7,A -85,B 0,C 180,E1 -18079.158,E2 -18079.158} C_VEL
LIN {X 0,Y 261.2,Z 692.862,A -85,B 0,C 180,E1 -18082.268,E2 -18082.268} C_VEL
LIN {X 0,Y 261.19,Z 694.822,A -85,B 0,C 180,E1 -18085.369,E2 -18085.369} C_VEL
LIN {X 0,Y 261.299,Z 695.595,A -85,B 0,C 180,E1 -18088.458,E2 -18088.458} C_VEL
LIN {X 0,Y 261.401,Z 695.512,A -85,B 0,C 180,E1 -18089.999,E2 -18089.999} C_VEL
LIN {X 0,Y 261.299,Z 694.395,A -85,B 0,C 180,E1 -18093.083,E2 -18093.083} C_VEL
LIN {X 0,Y 261.234,Z 692.039,A -85,B 0,C 180,E1 -18096.177,E2 -18096.177} C_VEL
LIN {X 0,Y 261.38,Z 688.388,A -85,B 0,C 180,E1 -18099.283,E2 -18099.283} C_VEL
LIN {X 0,Y 261.92,Z 683.354,A -85,B 0,C 180,E1 -18102.395,E2 -18102.395} C_VEL
LIN {X 0,Y 262.955,Z 676.802,A -85,B 0,C 180,E1 -18105.501,E2 -18105.501} C_VEL
LIN {X 0,Y 264.367,Z 669.705,A -85,B 0,C 180,E1 -18108.201,E2 -18108.201} C_VEL
LIN {X 0,Y 266.375,Z 661.139,A -85,B 0,C 180,E1 -18110.865,E2 -18110.865} C_VEL
LIN {X 0,Y 268.67,Z 651.189,A -85,B 0,C 180,E1 -18113.407,E2 -18113.407} C_VEL
LIN {X 0,Y 271.265,Z 640.163,A -85,B 0,C 180,E1 -18115.719,E2 -18115.719} C_VEL
LIN {X 0,Y 273.922,Z 628.637,A -85,B 0,C 180,E1 -18117.711,E2 -18117.711} C_VEL
LIN {X 0,Y 276.734,Z 616.14,A -85,B 0,C 180,E1 -18119.475,E2 -18119.475} C_VEL
LIN {X 0,Y 279.201,Z 603.906,A -85,B 0,C 180,E1 -18120.883,E2 -18120.883} C_VEL
LIN {X 0,Y 281.628,Z 589.45,A -85,B 0,C 180,E1 -18122.235,E2 -18122.235} C_VEL
LIN {X 0,Y 283.883,Z 574.197,A -85,B 0,C 180,E1 -18123.317,E2 -18123.317} C_VEL
LIN {X 0,Y 285.593,Z 559.077,A -85,B 0,C 180,E1 -18124.097,E2 -18124.097} C_VEL
LIN {X 0,Y 286.781,Z 543.633,A -85,B 0,C 180,E1 -18124.627,E2 -18124.627} C_VEL
LIN {X 0,Y 291.226,Z 447.426,A -85,B 0,C 180,E1 -18127.165,E2 -18127.165} C_VEL
LIN {X 0,Y 288.329,Z 427.41,A -85,B 0,C 180,E1 -18128.179,E2 -18128.179} C_VEL
LIN {X 0,Y 281.443,Z 411.269,A -85,B 0,C 180,E1 -18129.635,E2 -18129.635} C_VEL
LIN {X 0,Y 273.49,Z 394.359,A -85,B 0,C 180,E1 -18131.354,E2 -18131.354} C_VEL
LIN {X 0,Y 267.454,Z 382.097,A -85,B 0,C 180,E1 -18132.782,E2 -18132.782} C_VEL
LIN {X 0,Y 264.02,Z 370.38,A -85,B 0,C 180,E1 -18136.73,E2 -18136.73} C_VEL
LIN {X 0,Y 263.119,Z 367.325,A -85,B 0,C 180,E1 -18137.849,E2 -18137.849} C_VEL
LIN {X 0,Y 263.155,Z 367.322,A -85,B 0,C 180,E1 -18142.103,E2 -18142.103} C_VEL
LIN {X 0,Y 263.147,Z 367.325,A -85,B 0,C 180,E1 -18145.885,E2 -18145.885} C_VEL
LIN {X 0,Y 263.147,Z 367.335,A -85,B 0,C 180,E1 -18149.507,E2 -18149.507} C_VEL
LIN {X 0,Y 263.19,Z 367.327,A -85,B 0,C 180,E1 -18153.003,E2 -18153.003} C_VEL
LIN {X 0,Y 263.181,Z 367.326,A -85,B 0,C 180,E1 -18156.387,E2 -18156.387} C_VEL
LIN {X 0,Y 263.26,Z 367.317,A -85,B 0,C 180,E1 -18159.694,E2 -18159.694} C_VEL
LIN {X 0,Y 263.348,Z 367.308,A -85,B 0,C 180,E1 -18164.522,E2 -18164.522} C_VEL
LIN {X 0,Y 263.371,Z 367.277,A -85,B 0,C 180,E1 -18169.235,E2 -18169.235} C_VEL
LIN {X 0,Y 263.567,Z 367.272,A -85,B 0,C 180,E1 -18172.339,E2 -18172.339} C_VEL
LIN {X 0,Y 263.749,Z 367.242,A -85,B 0,C 180,E1 -18178.474,E2 -18178.474} C_VEL
LIN {X 0,Y 263.749,Z 367.254,A -85,B 0,C 180,E1 -18181.527,E2 -18181.527} C_VEL
LIN {X 0,Y 263.571,Z 367.263,A -85,B 0,C 180,E1 -18187.662,E2 -18187.662} C_VEL
LIN {X 0,Y 263.372,Z 367.303,A -85,B 0,C 180,E1 -18190.766,E2 -18190.766} C_VEL
LIN {X 0,Y 263.349,Z 367.291,A -85,B 0,C 180,E1 -18195.479,E2 -18195.479} C_VEL
LIN {X 0,Y 263.261,Z 367.315,A -85,B 0,C 180,E1 -18200.307,E2 -18200.307} C_VEL
LIN {X 0,Y 263.191,Z 367.306,A -85,B 0,C 180,E1 -18205.294,E2 -18205.294} C_VEL
LIN {X 0,Y 263.178,Z 367.324,A -85,B 0,C 180,E1 -18208.73,E2 -18208.73} C_VEL
LIN {X 0,Y 263.132,Z 367.332,A -85,B 0,C 180,E1 -18212.289,E2 -18212.289} C_VEL
LIN {X 0,Y 263.182,Z 367.319,A -85,B 0,C 180,E1 -18216.764,E2 -18216.764} C_VEL
LIN {X 0,Y 263.124,Z 367.328,A -85,B 0,C 180,E1 -18221.594,E2 -18221.594} C_VEL
LIN {X 0,Y 263.105,Z 367.333,A -85,B 0,C 180,E1 -18226.156,E2 -18226.156} C_VEL
LIN {X 0,Y 263.106,Z 367.33,A -85,B 0,C 180,E1 -18230.129,E2 -18230.129} C_VEL
LIN {X 0,Y 263.163,Z 367.328,A -85,B 0,C 180,E1 -18234.019,E2 -18234.019} C_VEL
LIN {X 0,Y 263.129,Z 367.326,A -85,B 0,C 180,E1 -18237.712,E2 -18237.712} C_VEL
LIN {X 0,Y 263.153,Z 367.33,A -85,B 0,C 180,E1 -18241.805,E2 -18241.805} C_VEL
LIN {X 0,Y 263.193,Z 367.321,A -85,B 0,C 180,E1 -18245.218,E2 -18245.218} C_VEL
LIN {X 0,Y 263.237,Z 367.311,A -85,B 0,C 180,E1 -18249.692,E2 -18249.692} C_VEL
LIN {X 0,Y 263.29,Z 367.308,A -85,B 0,C 180,E1 -18254.519,E2 -18254.519} C_VEL
LIN {X 0,Y 263.347,Z 367.305,A -85,B 0,C 180,E1 -18259.234,E2 -18259.234} C_VEL
LIN {X 0,Y 263.53,Z 367.281,A -85,B 0,C 180,E1 -18262.338,E2 -18262.338} C_VEL
LIN {X 0,Y 263.551,Z 367.28,A -85,B 0,C 180,E1 -18267.135,E2 -18267.135} C_VEL
LIN {X 0,Y 264.66,Z 370.242,A -85,B 0,C 180,E1 -18267.448,E2 -18267.448} C_VEL
LIN {X 0,Y 266.343,Z 372.483,A -85,B 0,C 180,E1 -18267.801,E2 -18267.801} C_VEL
LIN {X 0,Y 275.119,Z 387.457,A -85,B 0,C 180,E1 -18269.699,E2 -18269.699} C_VEL
LIN {X 0,Y 286.851,Z 409.323,A -85,B 0,C 180,E1 -18272.071,E2 -18272.071} C_VEL
LIN {X 0,Y 291.956,Z 419.991,A -85,B 0,C 180,E1 -18273.076,E2 -18273.076} C_VEL
LIN {X 0,Y 287.039,Z 521.076,A -85,B 0,C 180,E1 -18275.753,E2 -18275.753} C_VEL
LIN {X 0,Y 285.783,Z 536.706,A -85,B 0,C 180,E1 -18276.443,E2 -18276.443} C_VEL
LIN {X 0,Y 284.173,Z 551.6,A -85,B 0,C 180,E1 -18277.38,E2 -18277.38} C_VEL
LIN {X 0,Y 282.044,Z 566.378,A -85,B 0,C 180,E1 -18278.599,E2 -18278.599} C_VEL
LIN {X 0,Y 279.616,Z 580.847,A -85,B 0,C 180,E1 -18280.134,E2 -18280.134} C_VEL
LIN {X 0,Y 276.938,Z 594.257,A -85,B 0,C 180,E1 -18281.9,E2 -18281.9} C_VEL
LIN {X 0,Y 274.198,Z 606.866,A -85,B 0,C 180,E1 -18283.951,E2 -18283.951} C_VEL
LIN {X 0,Y 271.665,Z 617.815,A -85,B 0,C 180,E1 -18286.116,E2 -18286.116} C_VEL
LIN {X 0,Y 269.189,Z 627.955,A -85,B 0,C 180,E1 -18288.54,E2 -18288.54} C_VEL
LIN {X 0,Y 266.931,Z 637.157,A -85,B 0,C 180,E1 -18291.225,E2 -18291.225} C_VEL
LIN {X 0,Y 265.174,Z 644.524,A -85,B 0,C 180,E1 -18293.84,E2 -18293.84} C_VEL
LIN {X 0,Y 263.54,Z 651.567,A -85,B 0,C 180,E1 -18296.96,E2 -18296.96} C_VEL
LIN {X 0,Y 262.586,Z 656.404,A -85,B 0,C 180,E1 -18299.68,E2 -18299.68} C_VEL
LIN {X 0,Y 261.828,Z 660.211,A -85,B 0,C 180,E1 -18302.47,E2 -18302.47} C_VEL
LIN {X 0,Y 261.421,Z 662.235,A -85,B 0,C 180,E1 -18304.373,E2 -18304.373} C_VEL
LIN {X 0,Y 261.15,Z 663.821,A -85,B 0,C 180,E1 -18306.304,E2 -18306.304} C_VEL
LIN {X 0,Y 261.006,Z 665.085,A -85,B 0,C 180,E1 -18308.658,E2 -18308.658} C_VEL
LIN {X 0,Y 261.061,Z 665.702,A -85,B 0,C 180,E1 -18311.08,E2 -18311.08} C_VEL
LIN {X 0,Y 261.361,Z 665.413,A -85,B 0,C 180,E1 -18314.359,E2 -18314.359} C_VEL
LIN {X 0,Y 261.75,Z 664.568,A -85,B 0,C 180,E1 -18316.466,E2 -18316.466} C_VEL
LIN {X 0,Y 262.36,Z 663.147,A -85,B 0,C 180,E1 -18318.596,E2 -18318.596} C_VEL
LIN {X 0,Y 263.123,Z 661.08,A -85,B 0,C 180,E1 -18320.769,E2 -18320.769} C_VEL
LIN {X 0,Y 264.085,Z 658.383,A -85,B 0,C 180,E1 -18322.977,E2 -18322.977} C_VEL
LIN {X 0,Y 266.107,Z 652.964,A -85,B 0,C 180,E1 -18326.315,E2 -18326.315} C_VEL
LIN {X 0,Y 268.795,Z 645.771,A -85,B 0,C 180,E1 -18329.637,E2 -18329.637} C_VEL
LIN {X 0,Y 271.493,Z 638.603,A -85,B 0,C 180,E1 -18332.227,E2 -18332.227} C_VEL
LIN {X 0,Y 274.444,Z 630.606,A -85,B 0,C 180,E1 -18334.599,E2 -18334.599} C_VEL
LIN {X 0,Y 277.856,Z 620.842,A -85,B 0,C 180,E1 -18336.988,E2 -18336.988} C_VEL
LIN {X 0,Y 281.456,Z 609.492,A -85,B 0,C 180,E1 -18339.262,E2 -18339.262} C_VEL
LIN {X 0,Y 284.788,Z 598.265,A -85,B 0,C 180,E1 -18341.091,E2 -18341.091} C_VEL
LIN {X 0,Y 288.267,Z 585.293,A -85,B 0,C 180,E1 -18342.822,E2 -18342.822} C_VEL
LIN {X 0,Y 291.357,Z 571.694,A -85,B 0,C 180,E1 -18344.29,E2 -18344.29} C_VEL
LIN {X 0,Y 294.027,Z 557.861,A -85,B 0,C 180,E1 -18345.464,E2 -18345.464} C_VEL
LIN {X 0,Y 296.256,Z 542.675,A -85,B 0,C 180,E1 -18346.469,E2 -18346.469} C_VEL
LIN {X 0,Y 297.89,Z 527.65,A -85,B 0,C 180,E1 -18347.182,E2 -18347.182} C_VEL
LIN {X 0,Y 299.246,Z 508.623,A -85,B 0,C 180,E1 -18347.76,E2 -18347.76} C_VEL
LIN {X 0,Y 299.12,Z 502.86,A -85,B 0,C 180,E1 -18348.009,E2 -18348.009} C_VEL
LIN {X 0,Y 296.351,Z 484.415,A -85,B 0,C 180,E1 -18349.306,E2 -18349.306} C_VEL
LIN {X 0,Y 296.275,Z 478.654,A -85,B 0,C 180,E1 -18349.558,E2 -18349.558} C_VEL
LIN {X 0,Y 299.549,Z 430.304,A -85,B 0,C 180,E1 -18350.862,E2 -18350.862} C_VEL
LIN {X 0,Y 293.559,Z 418.991,A -85,B 0,C 180,E1 -18352.773,E2 -18352.773} C_VEL
LIN {X 0,Y 287.753,Z 409.346,A -85,B 0,C 180,E1 -18354.781,E2 -18354.781} C_VEL
LIN {X 0,Y 283.012,Z 402.112,A -85,B 0,C 180,E1 -18356.571,E2 -18356.571} C_VEL
LIN {X 0,Y 280.425,Z 398.638,A -85,B 0,C 180,E1 -18357.618,E2 -18357.618} C_VEL
LIN {X 0,Y 276.927,Z 393.651,A -85,B 0,C 180,E1 -18359.159,E2 -18359.159} C_VEL
LIN {X 0,Y 274.106,Z 389.643,A -85,B 0,C 180,E1 -18360.528,E2 -18360.528} C_VEL
LIN {X 0,Y 271.534,Z 386.329,A -85,B 0,C 180,E1 -18361.863,E2 -18361.863} C_VEL
LIN {X 0,Y 271.016,Z 385.287,A -85,B 0,C 180,E1 -18362.182,E2 -18362.182} C_VEL
LIN {X 0,Y 268.188,Z 382.836,A -85,B 0,C 180,E1 -18363.779,E2 -18363.779} C_VEL
LIN {X 0,Y 266.376,Z 379.907,A -85,B 0,C 180,E1 -18365.013,E2 -18365.013} C_VEL
LIN {X 0,Y 263.531,Z 377.732,A -85,B 0,C 180,E1 -18366.988,E2 -18366.988} C_VEL
LIN {X 0,Y 261.973,Z 374.782,A -85,B 0,C 180,E1 -18368.474,E2 -18368.474} C_VEL
LIN {X 0,Y 261.667,Z 374.151,A -85,B 0,C 180,E1 -18368.79,E2 -18368.79} C_VEL
LIN {X 0,Y 258.425,Z 372.449,A -85,B 0,C 180,E1 -18372.167,E2 -18372.167} C_VEL
LIN {X 0,Y 256.344,Z 368.882,A -85,B 0,C 180,E1 -18376.793,E2 -18376.793} C_VEL
LIN {X 0,Y 256.334,Z 368.984,A -85,B 0,C 180,E1 -18379.208,E2 -18379.208} C_VEL
LIN {X 0,Y 257.214,Z 371.092,A -85,B 0,C 180,E1 -18384.859,E2 -18384.859} C_VEL
LIN {X 0,Y 258.109,Z 372.471,A -85,B 0,C 180,E1 -18386.588,E2 -18386.588} C_VEL
LIN {X 0,Y 261.987,Z 378.18,A -85,B 0,C 180,E1 -18391.091,E2 -18391.091} C_VEL
LIN {X 0,Y 264.304,Z 381.075,A -85,B 0,C 180,E1 -18393.031,E2 -18393.031} C_VEL
LIN {X 0,Y 269.819,Z 388.915,A -85,B 0,C 180,E1 -18396.688,E2 -18396.688} C_VEL
LIN {X 0,Y 274.366,Z 395.823,A -85,B 0,C 180,E1 -18399.15,E2 -18399.15} C_VEL
LIN {X 0,Y 278.199,Z 401.963,A -85,B 0,C 180,E1 -18400.973,E2 -18400.973} C_VEL
LIN {X 0,Y 281.662,Z 407.843,A -85,B 0,C 180,E1 -18402.475,E2 -18402.475} C_VEL
LIN {X 0,Y 286.666,Z 416.773,A -85,B 0,C 180,E1 -18404.448,E2 -18404.448} C_VEL
LIN {X 0,Y 291.178,Z 426.022,A -85,B 0,C 180,E1 -18406.118,E2 -18406.118} C_VEL
LIN {X 0,Y 295.846,Z 436.691,A -85,B 0,C 180,E1 -18407.74,E2 -18407.74} C_VEL
LIN {X 0,Y 297.724,Z 441.733,A -85,B 0,C 180,E1 -18408.381,E2 -18408.381} C_VEL
LIN {X 0,Y 298.531,Z 452.133,A -85,B 0,C 180,E1 -18408.99,E2 -18408.99} C_VEL
LIN {X 0,Y 292.135,Z 546.712,A -85,B 0,C 180,E1 -18411.557,E2 -18411.557} C_VEL
LIN {X 0,Y 290.09,Z 563.17,A -85,B 0,C 180,E1 -18412.23,E2 -18412.23} C_VEL
LIN {X 0,Y 287.522,Z 578.216,A -85,B 0,C 180,E1 -18413.101,E2 -18413.101} C_VEL
LIN {X 0,Y 284.622,Z 591.531,A -85,B 0,C 180,E1 -18414.094,E2 -18414.094} C_VEL
LIN {X 0,Y 281.273,Z 605.055,A -85,B 0,C 180,E1 -18415.401,E2 -18415.401} C_VEL
LIN {X 0,Y 277.527,Z 618.408,A -85,B 0,C 180,E1 -18417.019,E2 -18417.019} C_VEL
LIN {X 0,Y 273.71,Z 630.809,A -85,B 0,C 180,E1 -18418.885,E2 -18418.885} C_VEL
LIN {X 0,Y 269.472,Z 643.163,A -85,B 0,C 180,E1 -18421.151,E2 -18421.151} C_VEL
LIN {X 0,Y 265.646,Z 654.252,A -85,B 0,C 180,E1 -18423.695,E2 -18423.695} C_VEL
LIN {X 0,Y 262.476,Z 663.511,A -85,B 0,C 180,E1 -18426.319,E2 -18426.319} C_VEL
LIN {X 0,Y 259.37,Z 672.298,A -85,B 0,C 180,E1 -18429.374,E2 -18429.374} C_VEL
LIN {X 0,Y 257.087,Z 679.431,A -85,B 0,C 180,E1 -18432.499,E2 -18432.499} C_VEL
LIN {X 0,Y 255.467,Z 685.102,A -85,B 0,C 180,E1 -18435.664,E2 -18435.664} C_VEL
LIN {X 0,Y 254.501,Z 689.439,A -85,B 0,C 180,E1 -18438.854,E2 -18438.854} C_VEL
LIN {X 0,Y 254.117,Z 692.536,A -85,B 0,C 180,E1 -18442.051,E2 -18442.051} C_VEL
LIN {X 0,Y 254.119,Z 694.444,A -85,B 0,C 180,E1 -18445.24,E2 -18445.24} C_VEL
LIN {X 0,Y 254.221,Z 695.169,A -85,B 0,C 180,E1 -18448.415,E2 -18448.415} C_VEL
LIN {X 0,Y 254.315,Z 695.078,A -85,B 0,C 180,E1 -18449.999,E2 -18449.999} C_VEL
LIN {X 0,Y 254.227,Z 693.915,A -85,B 0,C 180,E1 -18453.169,E2 -18453.169} C_VEL
LIN {X 0,Y 254.149,Z 691.499,A -85,B 0,C 180,E1 -18456.35,E2 -18456.35} C_VEL
LIN {X 0,Y 254.309,Z 687.785,A -85,B 0,C 180,E1 -18459.544,E2 -18459.544} C_VEL
LIN {X 0,Y 254.926,Z 682.685,A -85,B 0,C 180,E1 -18462.741,E2 -18462.741} C_VEL
LIN {X 0,Y 256.023,Z 676.058,A -85,B 0,C 180,E1 -18465.932,E2 -18465.932} C_VEL
LIN {X 0,Y 257.538,Z 668.882,A -85,B 0,C 180,E1 -18468.701,E2 -18468.701} C_VEL
LIN {X 0,Y 259.674,Z 660.227,A -85,B 0,C 180,E1 -18471.43,E2 -18471.43} C_VEL
LIN {X 0,Y 261.767,Z 651.409,A -85,B 0,C 180,E1 -18473.748,E2 -18473.748} C_VEL
LIN {X 0,Y 264.316,Z 640.965,A -85,B 0,C 180,E1 -18476.022,E2 -18476.022} C_VEL
LIN {X 0,Y 267.278,Z 628.523,A -85,B 0,C 180,E1 -18478.248,E2 -18478.248} C_VEL
LIN {X 0,Y 270.19,Z 616.074,A -85,B 0,C 180,E1 -18480.047,E2 -18480.047} C_VEL
LIN {X 0,Y 272.902,Z 603.015,A -85,B 0,C 180,E1 -18481.581,E2 -18481.581} C_VEL
LIN {X 0,Y 275.393,Z 588.552,A -85,B 0,C 180,E1 -18482.948,E2 -18482.948} C_VEL
LIN {X 0,Y 277.76,Z 573.162,A -85,B 0,C 180,E1 -18484.042,E2 -18484.042} C_VEL
LIN {X 0,Y 279.516,Z 557.79,A -85,B 0,C 180,E1 -18484.835,E2 -18484.835} C_VEL
LIN {X 0,Y 280.703,Z 541.755,A -85,B 0,C 180,E1 -18485.378,E2 -18485.378} C_VEL
LIN {X 0,Y 285.153,Z 448.354,A -85,B 0,C 180,E1 -18487.893,E2 -18487.893} C_VEL
LIN {X 0,Y 282.589,Z 430.098,A -85,B 0,C 180,E1 -18488.841,E2 -18488.841} C_VEL
LIN {X 0,Y 275.712,Z 414.028,A -85,B 0,C 180,E1 -18490.331,E2 -18490.331} C_VEL
LIN {X 0,Y 268.442,Z 398.409,A -85,B 0,C 180,E1 -18491.967,E2 -18491.967} C_VEL
LIN {X 0,Y 262.115,Z 385.894,A -85,B 0,C 180,E1 -18493.438,E2 -18493.438} C_VEL
LIN {X 0,Y 260.064,Z 381.674,A -85,B 0,C 180,E1 -18493.987,E2 -18493.987} C_VEL
LIN {X 0,Y 257.034,Z 371.427,A -85,B 0,C 180,E1 -18497.582,E2 -18497.582} C_VEL
LIN {X 0,Y 256.068,Z 368.205,A -85,B 0,C 180,E1 -18498.8,E2 -18498.8} C_VEL
LIN {X 0,Y 256.127,Z 368.202,A -85,B 0,C 180,E1 -18502.867,E2 -18502.867} C_VEL
LIN {X 0,Y 256.064,Z 368.204,A -85,B 0,C 180,E1 -18506.707,E2 -18506.707} C_VEL
LIN {X 0,Y 256.111,Z 368.21,A -85,B 0,C 180,E1 -18510.4,E2 -18510.4} C_VEL
LIN {X 0,Y 256.185,Z 368.196,A -85,B 0,C 180,E1 -18514.862,E2 -18514.862} C_VEL
LIN {X 0,Y 256.164,Z 368.202,A -85,B 0,C 180,E1 -18519.105,E2 -18519.105} C_VEL
LIN {X 0,Y 256.297,Z 368.185,A -85,B 0,C 180,E1 -18524.085,E2 -18524.085} C_VEL
LIN {X 0,Y 256.307,Z 368.155,A -85,B 0,C 180,E1 -18528.934,E2 -18528.934} C_VEL
LIN {X 0,Y 256.535,Z 368.147,A -85,B 0,C 180,E1 -18532.127,E2 -18532.127} C_VEL
LIN {X 0,Y 256.712,Z 368.117,A -85,B 0,C 180,E1 -18538.432,E2 -18538.432} C_VEL
LIN {X 0,Y 256.712,Z 368.131,A -85,B 0,C 180,E1 -18541.569,E2 -18541.569} C_VEL
LIN {X 0,Y 256.538,Z 368.139,A -85,B 0,C 180,E1 -18547.874,E2 -18547.874} C_VEL
LIN {X 0,Y 256.308,Z 368.184,A -85,B 0,C 180,E1 -18551.067,E2 -18551.067} C_VEL
LIN {X 0,Y 256.298,Z 368.167,A -85,B 0,C 180,E1 -18555.916,E2 -18555.916} C_VEL
LIN {X 0,Y 256.161,Z 368.203,A -85,B 0,C 180,E1 -18560.896,E2 -18560.896} C_VEL
LIN {X 0,Y 256.169,Z 368.181,A -85,B 0,C 180,E1 -18565.131,E2 -18565.131} C_VEL
LIN {X 0,Y 256.113,Z 368.205,A -85,B 0,C 180,E1 -18569.601,E2 -18569.601} C_VEL
LIN {X 0,Y 256.067,Z 368.202,A -85,B 0,C 180,E1 -18573.294,E2 -18573.294} C_VEL
LIN {X 0,Y 256.115,Z 368.203,A -85,B 0,C 180,E1 -18577.272,E2 -18577.272} C_VEL
LIN {X 0,Y 256.054,Z 368.209,A -85,B 0,C 180,E1 -18581.204,E2 -18581.204} C_VEL
LIN {X 0,Y 256.041,Z 368.211,A -85,B 0,C 180,E1 -18585.535,E2 -18585.535} C_VEL
LIN {X 0,Y 256.054,Z 368.212,A -85,B 0,C 180,E1 -18588.798,E2 -18588.798} C_VEL
LIN {X 0,Y 256.131,Z 368.2,A -85,B 0,C 180,E1 -18592.868,E2 -18592.868} C_VEL
LIN {X 0,Y 256.067,Z 368.208,A -85,B 0,C 180,E1 -18596.708,E2 -18596.708} C_VEL
LIN {X 0,Y 256.057,Z 368.213,A -85,B 0,C 180,E1 -18600.394,E2 -18600.394} C_VEL
LIN {X 0,Y 256.137,Z 368.197,A -85,B 0,C 180,E1 -18604.888,E2 -18604.888} C_VEL
LIN {X 0,Y 256.151,Z 368.194,A -85,B 0,C 180,E1 -18609.104,E2 -18609.104} C_VEL
LIN {X 0,Y 256.215,Z 368.189,A -85,B 0,C 180,E1 -18614.08,E2 -18614.08} C_VEL
LIN {X 0,Y 256.287,Z 368.183,A -85,B 0,C 180,E1 -18618.934,E2 -18618.934} C_VEL
LIN {X 0,Y 256.472,Z 368.158,A -85,B 0,C 180,E1 -18622.126,E2 -18622.126} C_VEL
LIN {X 0,Y 256.362,Z 368.203,A -85,B 0,C 180,E1 -18625.972,E2 -18625.972} C_VEL
LIN {X 0,Y 257.333,Z 370.952,A -85,B 0,C 180,E1 -18626.251,E2 -18626.251} C_VEL
LIN {X 0,Y 259.194,Z 373.341,A -85,B 0,C 180,E1 -18626.663,E2 -18626.663} C_VEL
LIN {X 0,Y 265.936,Z 384.275,A -85,B 0,C 180,E1 -18628.181,E2 -18628.181} C_VEL
LIN {X 0,Y 272.503,Z 396.23,A -85,B 0,C 180,E1 -18629.627,E2 -18629.627} C_VEL
LIN {X 0,Y 281.559,Z 413.059,A -85,B 0,C 180,E1 -18631.496,E2 -18631.496} C_VEL
LIN {X 0,Y 285.858,Z 422.265,A -85,B 0,C 180,E1 -18632.37,E2 -18632.37} C_VEL
LIN {X 0,Y 280.886,Z 521.463,A -85,B 0,C 180,E1 -18635.052,E2 -18635.052} C_VEL
LIN {X 0,Y 279.577,Z 537.004,A -85,B 0,C 180,E1 -18635.747,E2 -18635.747} C_VEL
LIN {X 0,Y 277.878,Z 552.144,A -85,B 0,C 180,E1 -18636.718,E2 -18636.718} C_VEL
LIN {X 0,Y 275.748,Z 566.505,A -85,B 0,C 180,E1 -18637.923,E2 -18637.923} C_VEL
LIN {X 0,Y 273.328,Z 580.592,A -85,B 0,C 180,E1 -18639.435,E2 -18639.435} C_VEL
LIN {X 0,Y 270.703,Z 593.557,A -85,B 0,C 180,E1 -18641.153,E2 -18641.153} C_VEL
LIN {X 0,Y 268.293,Z 604.253,A -85,B 0,C 180,E1 -18642.866,E2 -18642.866} C_VEL
LIN {X 0,Y 265.743,Z 615.063,A -85,B 0,C 180,E1 -18644.943,E2 -18644.943} C_VEL
LIN {X 0,Y 263.445,Z 624.324,A -85,B 0,C 180,E1 -18647.065,E2 -18647.065} C_VEL
LIN {X 0,Y 261.072,Z 633.502,A -85,B 0,C 180,E1 -18649.575,E2 -18649.575} C_VEL
LIN {X 0,Y 259.027,Z 641.757,A -85,B 0,C 180,E1 -18652.325,E2 -18652.325} C_VEL
LIN {X 0,Y 257.439,Z 648.039,A -85,B 0,C 180,E1 -18654.847,E2 -18654.847} C_VEL
LIN {X 0,Y 256.118,Z 653.959,A -85,B 0,C 180,E1 -18657.807,E2 -18657.807} C_VEL
LIN {X 0,Y 255.263,Z 658.19,A -85,B 0,C 180,E1 -18660.49,E2 -18660.49} C_VEL
LIN {X 0,Y 254.495,Z 661.856,A -85,B 0,C 180,E1 -18663.526,E2 -18663.526} C_VEL
LIN {X 0,Y 254.016,Z 664.444,A -85,B 0,C 180,E1 -18666.643,E2 -18666.643} C_VEL
LIN {X 0,Y 253.912,Z 665.776,A -85,B 0,C 180,E1 -18669.541,E2 -18669.541} C_VEL
LIN {X 0,Y 254.007,Z 666.186,A -85,B 0,C 180,E1 -18671.663,E2 -18671.663} C_VEL
LIN {X 0,Y 254.233,Z 665.984,A -85,B 0,C 180,E1 -18674.048,E2 -18674.048} C_VEL
LIN {X 0,Y 254.635,Z 665.189,A -85,B 0,C 180,E1 -18676.368,E2 -18676.368} C_VEL
LIN {X 0,Y 255.286,Z 663.838,A -85,B 0,C 180,E1 -18678.644,E2 -18678.644} C_VEL
LIN {X 0,Y 256.071,Z 661.895,A -85,B 0,C 180,E1 -18680.857,E2 -18680.857} C_VEL
LIN {X 0,Y 257.547,Z 658.147,A -85,B 0,C 180,E1 -18683.982,E2 -18683.982} C_VEL
LIN {X 0,Y 259.66,Z 652.818,A -85,B 0,C 180,E1 -18687.225,E2 -18687.225} C_VEL
LIN {X 0,Y 262.317,Z 646.197,A -85,B 0,C 180,E1 -18690.315,E2 -18690.315} C_VEL
LIN {X 0,Y 265.522,Z 638.157,A -85,B 0,C 180,E1 -18693.258,E2 -18693.258} C_VEL
LIN {X 0,Y 269.199,Z 628.627,A -85,B 0,C 180,E1 -18696.03,E2 -18696.03} C_VEL
LIN {X 0,Y 272.748,Z 618.654,A -85,B 0,C 180,E1 -18698.398,E2 -18698.398} C_VEL
LIN {X 0,Y 276.414,Z 607.647,A -85,B 0,C 180,E1 -18700.541,E2 -18700.541} C_VEL
LIN {X 0,Y 280.236,Z 595.262,A -85,B 0,C 180,E1 -18702.485,E2 -18702.485} C_VEL
